ABB RobotStudio station: project_station_1_34.rspag

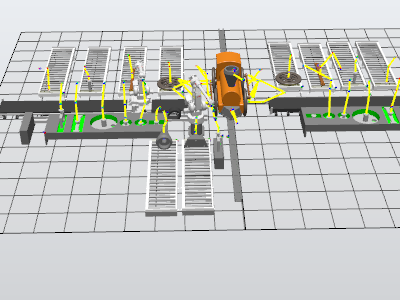
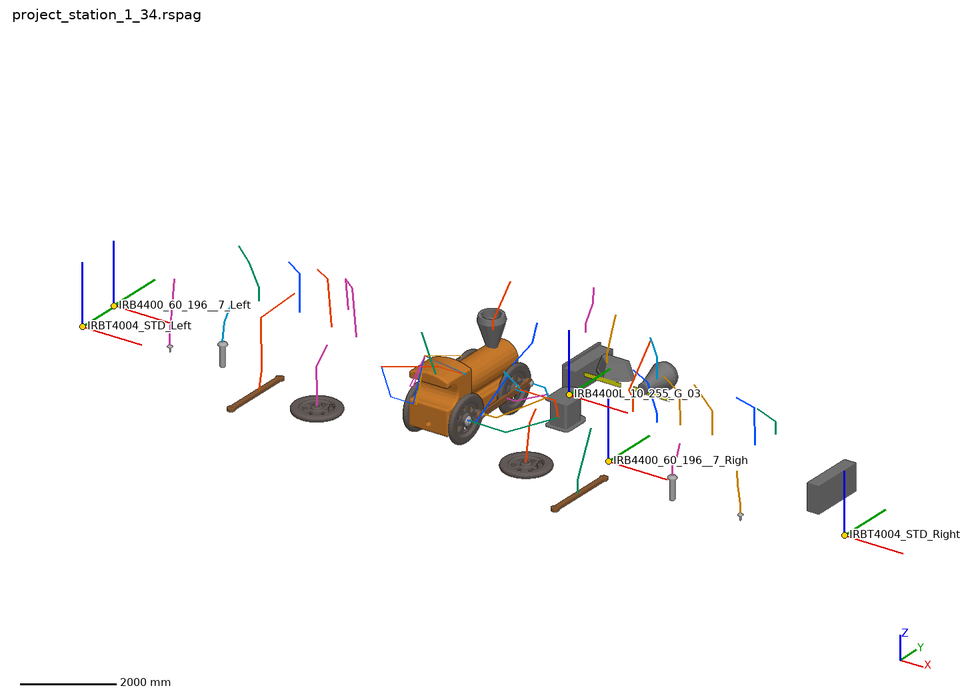
[picture v1: parts stored in the station drawn from their meshes, with robot base, taught points and paths (robot models come from the ABB library and are not in the file)]
--- station ---
Station project_station (saved by RobotStudio 24.1.10713.1)
Controller Controller2, task T_ROB1: task frame (RAPID world) sits at (1541.9, 2103.34, 619.07) mm, rotated rx 0 ry 0 rz 90 deg in the station
Controller Controller1, task T_ROB2: task frame (RAPID world) sits at (-8880.33, 560, 374.5) mm in the station
Controller Controller1, task T_ROB1: task frame (RAPID world) sits at (-8880.33, 560, 374.5) mm in the station
Controller Controller1
  mechanical unit ROB_1: IRB4400_60_196__7_Left, 6 joints, base frame (22.17, 0, 0) mm
  mechanical unit TRACK_1: IRBT4004_STD_Left, 1 joints, base frame (0, 0, 0) mm
  mechanical unit ROB_2: IRB4400_60_196__7_Right, 6 joints, base frame (17794.4, -138.17, 0) mm, rotated rx 0 ry 0 rz 180 deg
  mechanical unit TRACK_2: IRBT4004_STD_Right, 1 joints, base frame (17779.2, -146.88, 0) mm, rotated rx 0 ry 0 rz 180 deg
Controller Controller2
  mechanical unit ROB_1: IRB4400L_10_255_G_03, 6 joints, base frame (0, 0, 0) mm
Layout (positions relative to the parent item):
  - IRBT4004_STD_Right [mechanism] at (9294.37, 973.12, 0) mm, rotated rx 0 ry 0 rz 180 deg; joint values [5.175] (rad or m)
      links: Base, Link1
  - IRB4400_60_196__7_Left [mechanism, from %ABB.RobotStudio.Models.IRB4400%\IRB4400_60_196_G_03.rslib] at (-8880.33, 560, 374.5) mm; joint values [0, 0, 0, 0, 0.5236, 0] (rad or m)
  - IRB4400_60_196__7_Right [mechanism, from %ABB.RobotStudio.Models.IRB4400%\IRB4400_60_196_G_03.rslib] at (3723.87, 413.12, 374.5) mm, rotated rx 0 ry 0 rz 180 deg; joint values [-1.4312, -0.0428, -0.1313, 0, 1.1785, -0.0001] (rad or m)
  - IRBT4004_STD_Left [mechanism] at (-9275.83, 0, 0) mm; joint values [0] (rad or m)
      links: Base, Link1
  - Tool_Arm_Pin_Lift [mechanism, from Tool_geometries\my_Tool_Arm_Pin.rslib] at (-3735.45, 1947.72, 539.12) mm, rotated rx 180 ry 0 rz 180 deg
  - Tool_cow_catcher_Lift [mechanism, from Tool_geometries\my_Tool_Cow_Catcher.rslib] at (-3122.22, 1950.37, 611.02) mm, rotated rx 180 ry 0 rz 180 deg
  - Tool_Link_Right [mechanism, from Tool_geometries\my_Tool_Link.rslib] at (6128.18, 2244.28, 687.69) mm, rotated rx 180 ry -0.89 rz 180 deg
  - Tool_Stack_Right [mechanism, from Tool_geometries\my_Tool_Stack.rslib] at (733.33, 3848.22, 1135.13) mm, rotated rx 180 ry -0.01 rz -89.98 deg
  - Tool_Wheel_Right [mechanism, from Tool_geometries\my_Tool_Wheel.rslib] at (5126.19, 2141.41, 679.13) mm, rotated rx 180 ry 0 rz 180 deg
  - Tool_Axel_Pin_Lift [mechanism, from Tool_geometries\my_Too_Axel_pin.rslib] at (-4319.95, 1897.69, 635.99) mm, rotated rx 180 ry 0 rz 180 deg
  - Tool_Arm_Pin_Right [mechanism, from Tool_geometries\my_Tool_Arm_Pin.rslib] at (3680.28, 2224.13, 539.12) mm, rotated rx 180 ry 0 rz 180 deg
  - Tool_Axel_Pin_Right [mechanism, from Tool_geometries\my_Too_Axel_pin.rslib] at (4264.79, 2224.13, 633.5) mm, rotated rx 180 ry 0 rz 180 deg
  - Tool_cow_catcher_Right [mechanism, from Tool_geometries\my_Tool_Cow_Catcher.rslib] at (3068.05, 2237.38, 611.02) mm, rotated rx 180 ry 0 rz 180 deg
  - Tool_Link_Lift [mechanism, from Tool_geometries\my_Tool_Link.rslib] at (-6165.14, 1926.5, 700.28) mm, rotated rx 180 ry 0 rz 180 deg
  - Tool_Stack_Lift [mechanism, from Tool_geometries\my_Tool_Stack.rslib] at (-6789.17, 1963.76, 1135.13) mm, rotated rx 180 ry -0.01 rz 90.02 deg
  - Tool_Wheel_Lift [mechanism, from Tool_geometries\my_Tool_Wheel.rslib] at (-5181.37, 1991.55, 679.13) mm, rotated rx 180 ry 0 rz 180 deg
  - train_body [part] at (137.43, 399.25, 608.27) mm, rotated rx 0 ry 0 rz -90 deg, size 2750 x 1000 x 1362.5 mm
  - Wheel_Right_1 [part], size 1122.9 x 1119.7 x 250 mm
  - Wheel_Left_1 [part], size 1122.9 x 1119.7 x 250 mm
  - Table_tool_Right [part, from Tool_geometries\Stand_2.rslib] at (2653.05, 1565.95, 0) mm
  - Table_tool_Left [part, from Tool_geometries\Stand_2.rslib] at (-2708.23, 2555.9, 0) mm, rotated rx 0 ry 0 rz 180 deg
  - InFeeder_Right_1 [smart component, from Tool_geometries\my_InFeeder.rslib] at (2013.31, -295.59, 0) mm, rotated rx 0 ry 0 rz -90 deg
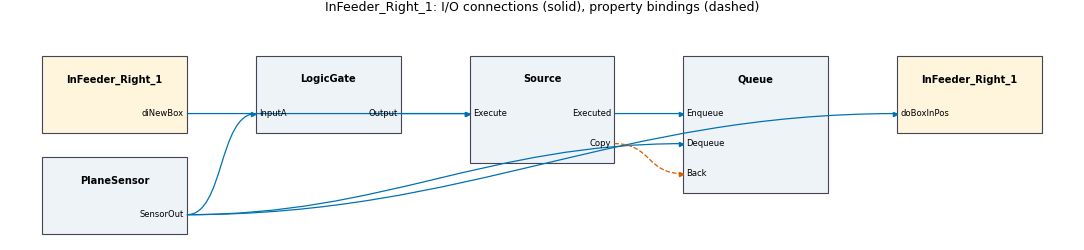
      connections:
        InFeeder_Right_1.diNewBox -> Source.Execute
        Source.Executed -> Queue.Enqueue
        PlaneSensor.SensorOut -> Queue.Dequeue
        PlaneSensor.SensorOut -> InFeeder_Right_1.doBoxInPos
        PlaneSensor.SensorOut -> LogicGate.InputA
        LogicGate.Output -> Source.Execute
        Source.Copy => Queue.Back
    - InFeeder [part, from Tool_geometries\my_InFeeder.rslib] at (-1070.62, 535.51, 0) mm
    - Source [smart component, from Components\Source.rslib] at (-1070.62, 535.51, 0) mm
        properties: Source=Wheel_Right_1; Copy=Wheel_Right_1_14; Parent=(none); Position=[0 0 0]; Orientation=[0 0 0]; Transient=false; PhysicsBehavior=-1
    - LinearMover [smart component, from Components\LinearMover.rslib] at (-1070.62, 535.51, 0) mm
        properties: Object=Queue; Direction=[0 1 0]; Speed=0.5; Reference=Global; ReferenceObject=(none)
    - Queue [smart component, from Components\Queue.rslib] at (-1070.62, 535.51, 0) mm
        properties: Back=Wheel_Right_1_14; Front=(none); Queue={1d023130-7791-4ef6-a898-f64e04810100};{8419fcdd-9884-4339-b140-c1e620e2220c};{d1e6a07f-8120-4cc8-bbc1-a0769f3691a2};{ab91239c-fc08-48bf-8341-3ec617d8a8b3}; NumberOfObjects=0
    - PlaneSensor [smart component, from Components\PlaneSensor.rslib] at (-1070.62, 535.51, 0) mm
        properties: Origin=[1.14 0.485 0.435]; Axis1=[0 0 0.1]; Axis2=[0 -0.93 0]; SensedPart=Wheel_Right_1_14; Tag=(none)
      - _sensorPart_ [part, from Tool_geometries\my_InFeeder.rslib]
    - LogicGate [smart component, from Components\LogicGate.rslib] at (-1070.62, 535.51, 0) mm
        properties: Operator=NOT; Delay=0
  - InFeeder_Right_2 [smart component, from Tool_geometries\my_InFeeder.rslib] at (3679.31, -295.59, 0) mm, rotated rx 0 ry 0 rz -90 deg
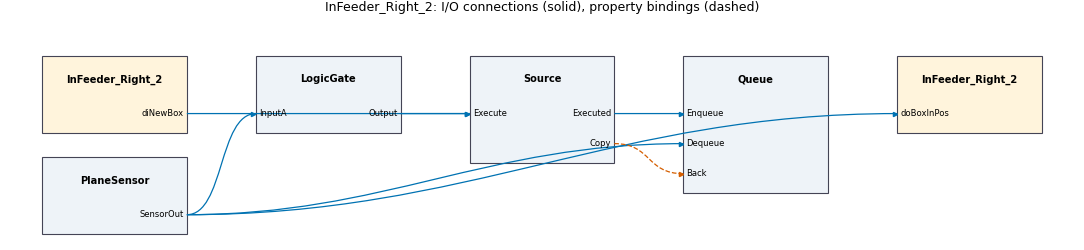
      connections:
        InFeeder_Right_2.diNewBox -> Source.Execute
        Source.Executed -> Queue.Enqueue
        PlaneSensor.SensorOut -> Queue.Dequeue
        PlaneSensor.SensorOut -> InFeeder_Right_2.doBoxInPos
        PlaneSensor.SensorOut -> LogicGate.InputA
        LogicGate.Output -> Source.Execute
        Source.Copy => Queue.Back
    - InFeeder [part, from Tool_geometries\my_InFeeder.rslib] at (-1070.62, 535.51, 0) mm
    - Source [smart component, from Components\Source.rslib] at (-1070.62, 535.51, 0) mm
        properties: Source=Link_Right_1; Copy=Link_Right_1_22; Parent=(none); Position=[0 0 0]; Orientation=[0 0 0]; Transient=false; PhysicsBehavior=-1
    - LinearMover [smart component, from Components\LinearMover.rslib] at (-1070.62, 535.51, 0) mm
        properties: Object=Queue; Direction=[0 1 0]; Speed=0.5; Reference=Global; ReferenceObject=(none)
    - Queue [smart component, from Components\Queue.rslib] at (-1070.62, 535.51, 0) mm
        properties: Back=Link_Right_1_22; Front=(none); Queue={ff46d1e0-f2c2-4271-a6c0-0c7e19cfd327};{f4dfb6bb-2350-47c6-830a-77889a19a4bb}; NumberOfObjects=0
    - PlaneSensor [smart component, from Components\PlaneSensor.rslib] at (-1070.62, 535.51, 0) mm
        properties: Origin=[1.14 0.485 0.435]; Axis1=[0 0 0.1]; Axis2=[0 -0.93 0]; SensedPart=Link_Right_1_22; Tag=(none)
      - _sensorPart_ [part, from Tool_geometries\my_InFeeder.rslib]
    - LogicGate [smart component, from Components\LogicGate.rslib] at (-1070.62, 535.51, 0) mm
        properties: Operator=NOT; Delay=0
  - InFeeder_Right_3 [smart component, from Tool_geometries\my_InFeeder.rslib] at (5345.31, -295.59, 0) mm, rotated rx 0 ry 0 rz -90 deg
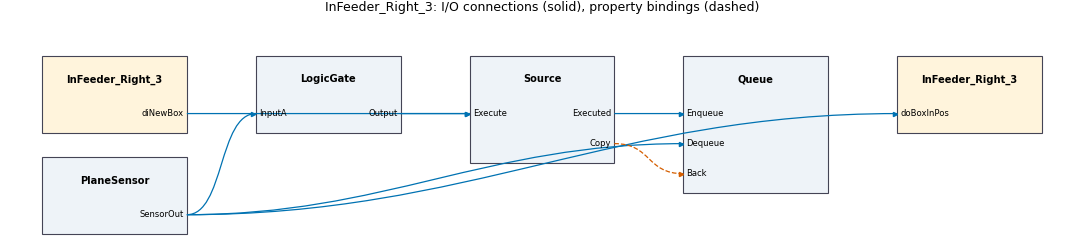
      connections:
        InFeeder_Right_3.diNewBox -> Source.Execute
        Source.Executed -> Queue.Enqueue
        PlaneSensor.SensorOut -> Queue.Dequeue
        PlaneSensor.SensorOut -> InFeeder_Right_3.doBoxInPos
        PlaneSensor.SensorOut -> LogicGate.InputA
        LogicGate.Output -> Source.Execute
        Source.Copy => Queue.Back
    - InFeeder [part, from Tool_geometries\my_InFeeder.rslib] at (-1070.62, 535.51, 0) mm
    - Source [smart component, from Components\Source.rslib] at (-1070.62, 535.51, 0) mm
        properties: Source=Axel_pin_Right_1; Copy=Axel_pin_Right_1_19; Parent=(none); Position=[0 0 0]; Orientation=[0 0 0]; Transient=false; PhysicsBehavior=-1
    - LinearMover [smart component, from Components\LinearMover.rslib] at (-1070.62, 535.51, 0) mm
        properties: Object=Queue; Direction=[0 1 0]; Speed=0.5; Reference=Global; ReferenceObject=(none)
    - Queue [smart component, from Components\Queue.rslib] at (-1070.62, 535.51, 0) mm
        properties: Back=Axel_pin_Right_1_19; Front=(none); Queue=; NumberOfObjects=0
    - PlaneSensor [smart component, from Components\PlaneSensor.rslib] at (-1070.62, 535.51, 0) mm
        properties: Origin=[1.14 0.485 0.435]; Axis1=[0 0 0.1]; Axis2=[0 -0.93 0]; SensedPart=Axel_pin_Right_1_19; Tag=(none)
      - _sensorPart_ [part, from Tool_geometries\my_InFeeder.rslib]
    - LogicGate [smart component, from Components\LogicGate.rslib] at (-1070.62, 535.51, 0) mm
        properties: Operator=NOT; Delay=0
  - InFeeder_Right_4 [smart component, from Tool_geometries\my_InFeeder.rslib] at (7011.31, -295.59, 0) mm, rotated rx 0 ry 0 rz -90 deg
      connections:
        InFeeder_Right_4.diNewBox -> Source.Execute
        Source.Executed -> Queue.Enqueue
        PlaneSensor.SensorOut -> Queue.Dequeue
        PlaneSensor.SensorOut -> InFeeder_Right_4.doBoxInPos
        PlaneSensor.SensorOut -> LogicGate.InputA
        LogicGate.Output -> Source.Execute
        Source.Copy => Queue.Back
    - InFeeder [part, from Tool_geometries\my_InFeeder.rslib] at (-1070.62, 535.51, 0) mm
    - Source [smart component, from Components\Source.rslib] at (-1070.62, 535.51, 0) mm
        properties: Source=Arm_pin_Right_1; Copy=Arm_pin_Right_1_24; Parent=(none); Position=[0 0 0]; Orientation=[0 0 0]; Transient=false; PhysicsBehavior=-1
    - LinearMover [smart component, from Components\LinearMover.rslib] at (-1070.62, 535.51, 0) mm
        properties: Object=Queue; Direction=[0 1 0]; Speed=0.5; Reference=Global; ReferenceObject=(none)
    - Queue [smart component, from Components\Queue.rslib] at (-1070.62, 535.51, 0) mm
        properties: Back=Arm_pin_Right_1_24; Front=(none); Queue=; NumberOfObjects=0
    - PlaneSensor [smart component, from Components\PlaneSensor.rslib] at (-1070.62, 535.51, 0) mm
        properties: Origin=[1.14 0.485 0.435]; Axis1=[0 0 0.1]; Axis2=[0 -0.93 0]; SensedPart=Arm_pin_Right_1_24; Tag=(none)
      - _sensorPart_ [part, from Tool_geometries\my_InFeeder.rslib]
    - LogicGate [smart component, from Components\LogicGate.rslib] at (-1070.62, 535.51, 0) mm
        properties: Operator=NOT; Delay=0
  - InFeeder_Left_1 [smart component, from Tool_geometries\my_InFeeder.rslib] at (-3038.95, -595.59, 0) mm, rotated rx 0 ry 0 rz -90 deg
      connections:
        InFeeder_Left_1.diNewBox -> Source.Execute
        Source.Executed -> Queue.Enqueue
        PlaneSensor.SensorOut -> Queue.Dequeue
        PlaneSensor.SensorOut -> InFeeder_Left_1.doBoxInPos
        PlaneSensor.SensorOut -> LogicGate.InputA
        LogicGate.Output -> Source.Execute
        Source.Copy => Queue.Back
    - InFeeder [part, from Tool_geometries\my_InFeeder.rslib] at (-1070.62, 535.51, 0) mm
    - Source [smart component, from Components\Source.rslib] at (-1070.62, 535.51, 0) mm
        properties: Source=Wheel_Left_1; Copy=Wheel_Left_1_13; Parent=(none); Position=[0 0 0]; Orientation=[0 0 0]; Transient=false; PhysicsBehavior=-1
    - LinearMover [smart component, from Components\LinearMover.rslib] at (-1070.62, 535.51, 0) mm
        properties: Object=Queue; Direction=[0 1 0]; Speed=0.5; Reference=Global; ReferenceObject=(none)
    - Queue [smart component, from Components\Queue.rslib] at (-1070.62, 535.51, 0) mm
        properties: Back=Wheel_Left_1_13; Front=(none); Queue=; NumberOfObjects=0
    - PlaneSensor [smart component, from Components\PlaneSensor.rslib] at (-1070.62, 535.51, 0) mm
        properties: Origin=[1.14 0.485 0.435]; Axis1=[0 0 0.1]; Axis2=[0 -0.93 0]; SensedPart=Wheel_Left_1_13; Tag=(none)
      - _sensorPart_ [part, from Tool_geometries\my_InFeeder.rslib]
    - LogicGate [smart component, from Components\LogicGate.rslib] at (-1070.62, 535.51, 0) mm
        properties: Operator=NOT; Delay=0
  - InFeeder_Left_2 [smart component, from Tool_geometries\my_InFeeder.rslib] at (-4426.95, -445.59, 0) mm, rotated rx 0 ry 0 rz -90 deg
      connections:
        InFeeder_Left_2.diNewBox -> Source.Execute
        Source.Executed -> Queue.Enqueue
        PlaneSensor.SensorOut -> Queue.Dequeue
        PlaneSensor.SensorOut -> InFeeder_Left_2.doBoxInPos
        PlaneSensor.SensorOut -> LogicGate.InputA
        LogicGate.Output -> Source.Execute
        Source.Copy => Queue.Back
    - InFeeder [part, from Tool_geometries\my_InFeeder.rslib] at (-1070.62, 535.51, 0) mm
    - Source [smart component, from Components\Source.rslib] at (-1070.62, 535.51, 0) mm
        properties: Source=Link_Left_1; Copy=Link_Left_1_18; Parent=(none); Position=[0 0 0]; Orientation=[0 0 0]; Transient=false; PhysicsBehavior=-1
    - LinearMover [smart component, from Components\LinearMover.rslib] at (-1070.62, 535.51, 0) mm
        properties: Object=Queue; Direction=[0 1 0]; Speed=0.5; Reference=Global; ReferenceObject=(none)
    - Queue [smart component, from Components\Queue.rslib] at (-1070.62, 535.51, 0) mm
        properties: Back=Link_Left_1_18; Front=(none); Queue={1ff3d472-21b5-4bb2-8564-f6cc722a728c}; NumberOfObjects=0
    - PlaneSensor [smart component, from Components\PlaneSensor.rslib] at (-1070.62, 535.51, 0) mm
        properties: Origin=[1.14 0.485 0.435]; Axis1=[0 0 0.1]; Axis2=[0 -0.93 0]; SensedPart=Link_Left_1_18; Tag=(none)
      - _sensorPart_ [part, from Tool_geometries\my_InFeeder.rslib]
    - LogicGate [smart component, from Components\LogicGate.rslib] at (-1070.62, 535.51, 0) mm
        properties: Operator=NOT; Delay=0
  - InFeeder_Left_3 [smart component, from Tool_geometries\my_InFeeder.rslib] at (-5792.95, -595.59, 0) mm, rotated rx 0 ry 0 rz -90 deg
      connections:
        InFeeder_Left_3.diNewBox -> Source.Execute
        Source.Executed -> Queue.Enqueue
        PlaneSensor.SensorOut -> Queue.Dequeue
        PlaneSensor.SensorOut -> InFeeder_Left_3.doBoxInPos
        PlaneSensor.SensorOut -> LogicGate.InputA
        LogicGate.Output -> Source.Execute
        Source.Copy => Queue.Back
    - InFeeder [part, from Tool_geometries\my_InFeeder.rslib] at (-1070.62, 535.51, 0) mm
    - Source [smart component, from Components\Source.rslib] at (-1070.62, 535.51, 0) mm
        properties: Source=Axel_pin_Left_1; Copy=Axel_pin_Left_1_16; Parent=(none); Position=[0 0 0]; Orientation=[0 0 0]; Transient=false; PhysicsBehavior=-1
    - LinearMover [smart component, from Components\LinearMover.rslib] at (-1070.62, 535.51, 0) mm
        properties: Object=Queue; Direction=[0 1 0]; Speed=0.5; Reference=Global; ReferenceObject=(none)
    - Queue [smart component, from Components\Queue.rslib] at (-1070.62, 535.51, 0) mm
        properties: Back=Axel_pin_Left_1_16; Front=(none); Queue={9023f18c-56cf-4535-be10-c416e51bdbb7};{c60a748b-6081-462f-837c-dfeccbfd19db};{920b546f-ac67-4257-bb71-08cb4a795493}; NumberOfObjects=0
    - PlaneSensor [smart component, from Components\PlaneSensor.rslib] at (-1070.62, 535.51, 0) mm
        properties: Origin=[1.14 0.485 0.435]; Axis1=[0 0 0.1]; Axis2=[0 -0.93 0]; SensedPart=Axel_pin_Left_1_16; Tag=(none)
      - _sensorPart_ [part, from Tool_geometries\my_InFeeder.rslib]
    - LogicGate [smart component, from Components\LogicGate.rslib] at (-1070.62, 535.51, 0) mm
        properties: Operator=NOT; Delay=0
  - InFeeder_Left_4 [smart component, from Tool_geometries\my_InFeeder.rslib] at (-7158.95, -595.59, 0) mm, rotated rx 0 ry 0 rz -90 deg
      connections:
        InFeeder_Left_4.diNewBox -> Source.Execute
        Source.Executed -> Queue.Enqueue
        PlaneSensor.SensorOut -> Queue.Dequeue
        PlaneSensor.SensorOut -> InFeeder_Left_4.doBoxInPos
        PlaneSensor.SensorOut -> LogicGate.InputA
        LogicGate.Output -> Source.Execute
        Source.Copy => Queue.Back
    - InFeeder [part, from Tool_geometries\my_InFeeder.rslib] at (-1070.62, 535.51, 0) mm
    - Source [smart component, from Components\Source.rslib] at (-1070.62, 535.51, 0) mm
        properties: Source=Arm_pin_Left_1; Copy=Arm_pin_Left_1_21; Parent=(none); Position=[0 0 0]; Orientation=[0 0 0]; Transient=false; PhysicsBehavior=-1
    - LinearMover [smart component, from Components\LinearMover.rslib] at (-1070.62, 535.51, 0) mm
        properties: Object=Queue; Direction=[0 1 0]; Speed=0.5; Reference=Global; ReferenceObject=(none)
    - Queue [smart component, from Components\Queue.rslib] at (-1070.62, 535.51, 0) mm
        properties: Back=Arm_pin_Left_1_21; Front=(none); Queue=; NumberOfObjects=0
    - PlaneSensor [smart component, from Components\PlaneSensor.rslib] at (-1070.62, 535.51, 0) mm
        properties: Origin=[1.14 0.485 0.435]; Axis1=[0 0 0.1]; Axis2=[0 -0.93 0]; SensedPart=Arm_pin_Left_1_21; Tag=(none)
      - _sensorPart_ [part, from Tool_geometries\my_InFeeder.rslib]
    - LogicGate [smart component, from Components\LogicGate.rslib] at (-1070.62, 535.51, 0) mm
        properties: Operator=NOT; Delay=0
  - Link_Right_1 [part] at (0, 300, 0) mm, size 186.8 x 1937.5 x 62.5 mm
  - train_tool_test [mechanism, from Tool_geometries\Train_Tool.rslib] at (0, 6532.17, 0) mm, rotated rx 0 ry 0 rz -90 deg; joint values [-0.5587, 0] (rad or m)
  - SC_AttachTool_Right [smart component] at (7697.63, 413.12, 2024.5) mm, rotated rx 180 ry 60 rz 0 deg
      signals: DI diAttachTool
      connections:
        SC_AttachTool_Right.diAttachTool -> ClosestObject.Execute
        ClosestObject.Executed -> Attacher.Execute
        SC_AttachTool_Right.diAttachTool -> LogicGate.InputA
        LogicGate.Output -> Detacher.Execute
        ClosestObject.ClosestObject => Attacher.Child
        Attacher.Child => Detacher.Child
    - Attacher [smart component, from Components\Attacher.rslib]
        properties: Parent=IRB4400_60_196__7_Right; Flange=0; Child=Tool_Arm_Pin_Right; Mount=false; Offset=[0 0 0]; Orientation=[0 0 0]
    - Detacher [smart component, from Components\Detacher.rslib]
        properties: Child=Tool_Arm_Pin_Right; KeepPosition=true
    - ClosestObject [smart component, from Components\ClosestObject.rslib]
        properties: ReferenceObject=IRB4400_60_196__7_Right; ReferencePoint=[7.697628 0.41312 2.0245]; RootObject=(none); ClosestObject=Tool_Arm_Pin_Right; ClosestPart=Tool_Arm_pin; Distance=0
    - LogicGate [smart component, from Components\LogicGate.rslib]
        properties: Operator=NOT; Delay=0
  - Axel_pin_Left_1 [part] at (1364.35, 150, 0) mm, size 211 x 211 x 562.7 mm
  - Arm_pin_Left_1 [part], size 126 x 125.8 x 162.5 mm
  - Link_Left_1 [part], size 186.8 x 1937.5 x 62.5 mm
  - SC_AttachTool_left [smart component] at (-8447.37, 1113.95, 2155.74) mm, rotated rx 180 ry 60 rz -130.35 deg
      signals: DI diAT_Left
      connections:
        SC_AttachTool_left.diAT_Left -> ClosestObject.Execute
        ClosestObject.Executed -> Attacher.Execute
        SC_AttachTool_left.diAT_Left -> LogicGate.InputA
        LogicGate.Output -> Detacher.Execute
        ClosestObject.ClosestObject => Attacher.Child
        Attacher.Child => Detacher.Child
    - Attacher [smart component, from Components\Attacher.rslib]
        properties: Parent=IRB4400_60_196__7_Left; Flange=0; Child=Tool_Arm_Pin_Lift; Mount=false; Offset=[0 0 0]; Orientation=[0 0 0]
    - Detacher [smart component, from Components\Detacher.rslib]
        properties: Child=Tool_Arm_Pin_Lift; KeepPosition=true
    - ClosestObject [smart component, from Components\ClosestObject.rslib]
        properties: ReferenceObject=IRB4400_60_196__7_Left; ReferencePoint=[-7.679085 0.56 2.0245]; RootObject=(none); ClosestObject=Tool_Arm_Pin_Lift; ClosestPart=Tool_Arm_pin; Distance=0
    - LogicGate [smart component, from Components\LogicGate.rslib]
        properties: Operator=NOT; Delay=0
  - Axel_pin_Right_1 [part], size 211 x 211 x 562.7 mm
  - Arm_pin_Right_1 [part], size 126 x 125.8 x 162.5 mm
  - RobotStand2400H620 [part] at (1512.32, 2162.24, 0) mm, size 600 x 830 x 620 mm
  - IRB4400L_10_255_G_03 [mechanism, from %ABB.RobotStudio.Models.IRB4400%\IRB4400L_10_255_G_03.rslib] at (1541.9, 2103.34, 619.07) mm, rotated rx 0 ry 0 rz 90 deg; joint values [0.3142, 0, 0, 0, 0.9774, 0] (rad or m)
  - SC_InFeeder [smart component, from Solutions\SC_InFeeder.rslib] at (2782.92, 2208.74, 0) mm, rotated rx 0 ry 0 rz 90 deg
      connections:
        SC_InFeeder.diNewBox -> Source.Execute
        Source.Executed -> Queue.Enqueue
        PlaneSensor.SensorOut -> Queue.Dequeue
        PlaneSensor.SensorOut -> SC_InFeeder.doBoxInPos
        PlaneSensor.SensorOut -> LogicGate.InputA
        LogicGate.Output -> Source.Execute
        Source.Copy => Queue.Back
    - InFeeder [part, from Solutions\SC_InFeeder.rslib]
    - Source [smart component, from Components\Source.rslib]
        properties: Source=Stack_tutorial; Copy=Stack_tutorial_26; Parent=(none); Position=[0 0 0]; Orientation=[0 0 0]; Transient=false; PhysicsBehavior=-1
    - LinearMover [smart component, from Components\LinearMover.rslib]
        properties: Object=Queue; Direction=[0 -1 0]; Speed=0.5; Reference=Global; ReferenceObject=(none)
    - Queue [smart component, from Components\Queue.rslib]
        properties: Back=Stack_tutorial_26; Front=(none); Queue=; NumberOfObjects=0
    - PlaneSensor [smart component, from Components\PlaneSensor.rslib]
        properties: Origin=[1.14 0.485 0.435]; Axis1=[0 0 0.1]; Axis2=[0 -0.93 0]; SensedPart=Stack_tutorial_26; Tag=(none)
      - _sensorPart_ [part], size 0 x 930 x 100 mm
    - LogicGate [smart component, from Components\LogicGate.rslib]
        properties: Operator=NOT; Delay=0
  - SC_InFeeder_1 [smart component, from Solutions\SC_InFeeder.rslib] at (1551.58, 2174.69, 0) mm, rotated rx 0 ry 0 rz 90 deg
      connections:
        SC_InFeeder_1.diNewBox -> Source.Execute
        Source.Executed -> Queue.Enqueue
        PlaneSensor.SensorOut -> Queue.Dequeue
        PlaneSensor.SensorOut -> SC_InFeeder_1.doBoxInPos
        PlaneSensor.SensorOut -> LogicGate.InputA
        LogicGate.Output -> Source.Execute
        Source.Copy => Queue.Back
    - InFeeder [part, from Solutions\SC_InFeeder.rslib]
    - Source [smart component, from Components\Source.rslib]
        properties: Source=Cow_Catcher; Copy=Cow_Catcher_25; Parent=(none); Position=[0 0 0]; Orientation=[0 0 0]; Transient=false; PhysicsBehavior=-1
    - LinearMover [smart component, from Components\LinearMover.rslib]
        properties: Object=Queue; Direction=[0 -1 0]; Speed=0.5; Reference=Global; ReferenceObject=(none)
    - Queue [smart component, from Components\Queue.rslib]
        properties: Back=Cow_Catcher_25; Front=(none); Queue=; NumberOfObjects=0
    - PlaneSensor [smart component, from Components\PlaneSensor.rslib]
        properties: Origin=[1.14 0.485 0.435]; Axis1=[0 0 0.1]; Axis2=[0 -0.93 0]; SensedPart=Cow_Catcher_25; Tag=(none)
      - _sensorPart_ [part], size 0 x 930 x 100 mm
    - LogicGate [smart component, from Components\LogicGate.rslib]
        properties: Operator=NOT; Delay=0
  - Cow_Catcher [part], size 900 x 562.5 x 375 mm
  - Stack_tutorial [part], size 625 x 875 x 623.8 mm
  - SmartComponent_1 [smart component] at (1001.89, 3765.34, 2268.6) mm, rotated rx -180 ry 34 rz -72 deg
      signals: DI di_Rob3_at_tool
      connections:
        SmartComponent_1.di_Rob3_at_tool -> ClosestObject.Execute
        ClosestObject.Executed -> Attacher.Execute
        SmartComponent_1.di_Rob3_at_tool -> LogicGate.InputA
        LogicGate.Output -> Detacher.Execute
        ClosestObject.ClosestObject => Attacher.Child
        Attacher.Child => Detacher.Child
    - Attacher [smart component, from Components\Attacher.rslib]
        properties: Parent=IRB4400L_10_255_G_03; Flange=0; Child=Tool_Stack_Right; Mount=false; Offset=[0 0 0]; Orientation=[0 0 0]
    - Detacher [smart component, from Components\Detacher.rslib]
        properties: Child=Tool_Stack_Right; KeepPosition=true
    - ClosestObject [smart component, from Components\ClosestObject.rslib] at (0, 0.07, 0.19) mm, rotated rx 0 ry 0 rz 0.01 deg
        properties: ReferenceObject=IRB4400L_10_255_G_03; ReferencePoint=[1.623149 3.935855 2.269225]; RootObject=(none); ClosestObject=Tool_Stack_Right; ClosestPart=Tool_Stack_tutorial; Distance=0
    - LogicGate [smart component, from Components\LogicGate.rslib]
        properties: Operator=NOT; Delay=0
  - Tool_Stack [mechanism, from Tool_geometries\my_Tool_Stack.rslib] at (6727.73, 2146.19, 1135.13) mm, rotated rx 180 ry -0.01 rz -89.98 deg
  - Part_1 [part] at (7983.1, 1490.43, 0) mm, size 300 x 1350 x 650 mm
  - Part_10 [part] at (543.39, 3269.91, 0) mm, size 348.3 x 1331.4 x 570 mm
  - Axel_pin_Left_1_1 [part] at (501.33, -5711.63, 5481.38) mm, rotated rx 90 ry 0 rz -90 deg, size 211 x 211 x 562.7 mm
  - Arm_pin_Left_1_2 [part] at (-187.19, 6322.39, -3373.2) mm, rotated rx -88 ry -0.94 rz 89.66 deg, size 126 x 125.8 x 162.5 mm
  - Stack_tutorial_3 [part] at (191.58, -1196.82, -5198.95) mm, rotated rx 89.7 ry -2.42 rz 106.93 deg, size 625 x 875 x 623.8 mm
  - Cow_Catcher_4 [part] at (2358.03, 9034.46, -915.07) mm, rotated rx 8.93 ry 3.16 rz 175.56 deg, size 900 x 562.5 x 375 mm
  - Link_Left_1_5 [part] at (-36.44, -4252.23, -2713.27) mm, rotated rx 99.73 ry 90 rz -80.27 deg, size 186.8 x 1937.5 x 62.5 mm
  - Wheel_Right_1_6 [part] at (297.93, -1737.55, 5267.12) mm, rotated rx 91.04 ry -5.67 rz 89.75 deg, size 1122.9 x 1119.7 x 250 mm
  - Link_Right_1_7 [part] at (436, -3607.65, -3457.42) mm, rotated rx -88.02 ry -88 rz -91.77 deg, size 186.8 x 1937.5 x 62.5 mm
  - Axel_pin_Right_1_8 [part] at (-147.05, -5745.67, 2902.14) mm, rotated rx 90 ry -20 rz 90 deg, size 211 x 211 x 562.7 mm
  - Arm_pin_Right_1_9 [part] at (1185.67, -6952.34, -808.64) mm, rotated rx 88.67 ry -40.63 rz 96.05 deg, size 126 x 125.8 x 162.5 mm
  - Wheel_Left_1_10 [part] at (65.04, 4540.99, 1028.75) mm, rotated rx -90 ry -62 rz 90 deg, size 1122.9 x 1119.7 x 250 mm
  - Wheel_Left_1_11 [part] at (65.04, 6286.67, 1028.75) mm, rotated rx -90 ry -62 rz 90 deg, size 1122.9 x 1119.7 x 250 mm
  - Wheel_Right_1_12 [part] at (374.22, -3437.13, 5308.69) mm, rotated rx 93.56 ry -5.2 rz 87.1 deg, size 1122.9 x 1119.7 x 250 mm
  - Wheel_Left_1_13 [part] at (0, 3132, 0) mm, size 1122.9 x 1119.7 x 250 mm
  - Wheel_Right_1_14 [part] at (0, 3756, 0) mm, size 1122.9 x 1119.7 x 250 mm
  - Axel_pin_Left_1_15 [part] at (501.09, -3965.51, 5481.38) mm, rotated rx 90 ry 0 rz -90 deg, size 211 x 211 x 562.7 mm
  - Axel_pin_Left_1_16 [part] at (0, 3900, 0) mm, size 211 x 211 x 562.7 mm
  - Axel_pin_Right_1_17 [part] at (-152.97, -7511.91, 2881.93) mm, rotated rx 90 ry -20 rz 90 deg, size 211 x 211 x 562.7 mm
  - Link_Left_1_18 [part] at (0, 3312, 0) mm, size 186.8 x 1937.5 x 62.5 mm
  - Axel_pin_Right_1_19 [part] at (0, 3900, 0) mm, size 211 x 211 x 562.7 mm
  - Arm_pin_Left_1_20 [part] at (-187.19, 8072.39, -3373.2) mm, rotated rx -88 ry -0.94 rz 89.66 deg, size 126 x 125.8 x 162.5 mm
  - Arm_pin_Left_1_21 [part] at (0, 3960, 0) mm, size 126 x 125.8 x 162.5 mm
  - Link_Right_1_22 [part] at (0, 3132, 0) mm, size 186.8 x 1937.5 x 62.5 mm
  - Arm_pin_Right_1_23 [part] at (1192.07, -8711.93, -803.85) mm, rotated rx 88.67 ry -40.63 rz 96.05 deg, size 126 x 125.8 x 162.5 mm
  - Arm_pin_Right_1_24 [part] at (0, 3912, 0) mm, size 126 x 125.8 x 162.5 mm
  - Cow_Catcher_25 [part] at (0, -3876, 0) mm, size 900 x 562.5 x 375 mm
  - Stack_tutorial_26 [part] at (0, -3564, 0) mm, size 625 x 875 x 623.8 mm
Attachment: IRB4400_60_196__7_Left is attached to IRBT4004_STD_Left / Link1
Attachment: stand_tool_Right is attached to Table_tool_Right
Attachment: stand_tool_Left is attached to Table_tool_Left
Attachment: Tool_cow_catcher_Lift is attached to Table_tool_Left
Attachment: InFeWOb_Right_1 is attached to InFeeder
Attachment: InFeWOb_Right_2 is attached to InFeeder
Attachment: InFeWOb_Right_3 is attached to InFeeder
Attachment: InFeWOb_Right_4 is attached to InFeeder
Attachment: Link_Right_1 is attached to InFeeder_Right_2
Attachment: InFeWOb_Lift_1 is attached to InFeeder
Attachment: InFeWOb_Lift_3 is attached to InFeeder
Attachment: InFeWOb_Lift_2 is attached to InFeeder
Attachment: InFeWOb_Lift_4 is attached to InFeeder
Attachment: TrRiFcWOb is attached to train_body
Attachment: TrLeFcWob is attached to train_body
Attachment: Arm_pin_Left_1 is attached to InFeeder_Left_3
Attachment: Axel_pin_Left_1 is attached to InFeeder_Left_2
Attachment: Link_Left_1 is attached to InFeeder_Left_4
Attachment: Wheel_Left_1 is attached to InFeeder_Left_1
Attachment: Axel_pin_Right_1 is attached to InFeeder_Right_3
Attachment: Arm_pin_Right_1 is attached to InFeeder_Right_4
Attachment: IRB4400_60_196__7_Right is attached to IRBT4004_STD_Right / Link1
Attachment: WokOb_feed_1_Caw is attached to InFeeder
Attachment: WokOb_feed is attached to InFeeder
Attachment: WokOb_tarin_Front is attached to train_body
Attachment: WokOb_Train_Top is attached to train_body
Attachment: SmartComponent_1 is attached to IRB4400L_10_255_G_03 / Link6
Attachment: Cow_Catcher is attached to SC_InFeeder_1
Attachment: IRB4400L_10_255_G_03 is attached to RobotStand2400H620
Attachment: WorOb_Stacl_Rb3 is attached to Part_10
EventTableEntry 6118: Group=, Trigger=diAttachTool 6119, Actions=[EventTableActionAttach 6120], Comment=, ActivationMode=2, Cyclic=false
EventTableTriggerIO 6119: IOValue=[1], IRC5Controller=? -1, Operator=0, SignalSource=Controller1 3715
EventTableActionAttach 6120: AttachmentParent=IRB4400_60_196__7_Right 3583, AttachmentChild=? -1, MountObject=false, Offset=[X=1, Y=0, Z=0, W=0, X=0, Y=1, Z=0, W=0, X=0, Y=0, Z=1, W=0, X=0, Y=0, Z=0, W=1], FlangeIndext=0, FindNearest=true
EventTableEntry 6121: Group=, Trigger=diAttachTool 6122, Actions=[EventTableActionDetach 6123], Comment=, ActivationMode=2, Cyclic=false
EventTableTriggerIO 6122: IOValue=[0], IRC5Controller=? -1, Operator=0, SignalSource=Controller1 3715
EventTableActionDetach 6123: AttachmentParent=IRB4400_60_196__7_Right 3583, AttachmentChild=? -1
EventTableEntry 8584: Group=, Trigger=doAttachTool 8585, Actions=[EventTableActionAttach 8586], Comment=, ActivationMode=2, Cyclic=false
EventTableTriggerIO 8585: IOValue=[1], IRC5Controller=? -1, Operator=0, SignalSource=Controller1 3715
EventTableActionAttach 8586: AttachmentParent=IRB4400_60_196__7_Left 2378, AttachmentChild=? -1, MountObject=false, Offset=[X=1, Y=0, Z=0, W=0, X=0, Y=1, Z=0, W=0, X=0, Y=0, Z=1, W=0, X=0, Y=0, Z=0, W=1], FlangeIndext=0, FindNearest=true
EventTableEntry 8587: Group=, Trigger=doAttachTool 8588, Actions=[EventTableActionDetach 8589], Comment=, ActivationMode=2, Cyclic=false
EventTableTriggerIO 8588: IOValue=[0], IRC5Controller=? -1, Operator=0, SignalSource=Controller1 3715
EventTableActionDetach 8589: AttachmentParent=IRB4400_60_196__7_Left 2378, AttachmentChild=? -1
EventTableEntry 10457: Group=, Trigger=doAtWhRi 10458, Actions=[EventTableActionAttach 10459], Comment=, ActivationMode=2, Cyclic=false
EventTableTriggerIO 10458: IOValue=[1], IRC5Controller=? -1, Operator=0, SignalSource=Controller1 3715
EventTableActionAttach 10459: AttachmentParent=Tool_Wheel_Right 3673, AttachmentChild=? -1, MountObject=false, Offset=[X=1, Y=0, Z=0, W=0, X=0, Y=1, Z=0, W=0, X=0, Y=0, Z=1, W=0, X=0, Y=0, Z=0, W=1], FlangeIndext=0, FindNearest=true
EventTableEntry 10462: Group=, Trigger=doAtWhRi 10463, Actions=[EventTableActionDetach 10464], Comment=, ActivationMode=2, Cyclic=false
EventTableTriggerIO 10463: IOValue=[0], IRC5Controller=? -1, Operator=0, SignalSource=Controller1 3715
EventTableActionDetach 10464: AttachmentParent=Tool_Wheel_Right 3673, AttachmentChild=? -1
EventTableEntry 10559: Group=, Trigger=Att_link 10560, Actions=[EventTableActionAttach 10561], Comment=, ActivationMode=2, Cyclic=false
EventTableTriggerIO 10560: IOValue=[1], IRC5Controller=? -1, Operator=0, SignalSource=Controller1 3715
EventTableActionAttach 10561: AttachmentParent=Tool_Link_Right 3667, AttachmentChild=? -1, MountObject=false, Offset=[X=1, Y=0, Z=0, W=0, X=0, Y=1, Z=0, W=0, X=0, Y=0, Z=1, W=0, X=0, Y=0, Z=0, W=1], FlangeIndext=0, FindNearest=true
EventTableEntry 10562: Group=, Trigger=Att_link 10563, Actions=[EventTableActionDetach 10564], Comment=, ActivationMode=2, Cyclic=false
EventTableTriggerIO 10563: IOValue=[0], IRC5Controller=? -1, Operator=0, SignalSource=Controller1 3715
EventTableActionDetach 10564: AttachmentParent=Tool_Link_Right 3667, AttachmentChild=? -1
EventTableEntry 13658: Group=, Trigger=doAt_Wh_Left 13659, Actions=[EventTableActionAttach 13660], Comment=, ActivationMode=2, Cyclic=false
EventTableTriggerIO 13659: IOValue=[1], IRC5Controller=? -1, Operator=0, SignalSource=Controller1 3715
EventTableActionAttach 13660: AttachmentParent=Tool_Wheel_Lift 3694, AttachmentChild=? -1, MountObject=false, Offset=[X=1, Y=0, Z=0, W=0, X=0, Y=1, Z=0, W=0, X=0, Y=0, Z=1, W=0, X=0, Y=0, Z=0, W=1], FlangeIndext=0, FindNearest=true
EventTableEntry 13661: Group=, Trigger=doAt_Wh_Left 13662, Actions=[EventTableActionDetach 13663], Comment=, ActivationMode=2, Cyclic=false
EventTableTriggerIO 13662: IOValue=[0], IRC5Controller=? -1, Operator=0, SignalSource=Controller1 3715
EventTableActionDetach 13663: AttachmentParent=Tool_Wheel_Lift 3694, AttachmentChild=? -1
EventTableEntry 13664: Group=, Trigger=doAt_Link_Left 13665, Actions=[EventTableActionAttach 13666], Comment=, ActivationMode=2, Cyclic=false
EventTableTriggerIO 13665: IOValue=[1], IRC5Controller=? -1, Operator=0, SignalSource=Controller1 3715
EventTableActionAttach 13666: AttachmentParent=Tool_Link_Lift 3688, AttachmentChild=? -1, MountObject=false, Offset=[X=1, Y=0, Z=0, W=0, X=0, Y=1, Z=0, W=0, X=0, Y=0, Z=1, W=0, X=0, Y=0, Z=0, W=1], FlangeIndext=0, FindNearest=true
EventTableEntry 13667: Group=, Trigger=doAt_Link_Left 13668, Actions=[EventTableActionDetach 13669], Comment=, ActivationMode=2, Cyclic=false
EventTableTriggerIO 13668: IOValue=[0], IRC5Controller=? -1, Operator=0, SignalSource=Controller1 3715
EventTableActionDetach 13669: AttachmentParent=Tool_Link_Lift 3688, AttachmentChild=? -1
EventTableEntry 13670: Group=, Trigger=doAt_AxelP_Left 13671, Actions=[EventTableActionAttach 13672], Comment=, ActivationMode=2, Cyclic=false
EventTableTriggerIO 13671: IOValue=[1], IRC5Controller=? -1, Operator=0, SignalSource=Controller1 3715
EventTableActionAttach 13672: AttachmentParent=Tool_Axel_Pin_Lift 3676, AttachmentChild=? -1, MountObject=false, Offset=[X=1, Y=0, Z=0, W=0, X=0, Y=1, Z=0, W=0, X=0, Y=0, Z=1, W=0, X=0, Y=0, Z=0, W=1], FlangeIndext=0, FindNearest=true
EventTableEntry 13673: Group=, Trigger=doAt_AxelP_Left 13674, Actions=[EventTableActionDetach 13675], Comment=, ActivationMode=2, Cyclic=false
EventTableTriggerIO 13674: IOValue=[0], IRC5Controller=? -1, Operator=0, SignalSource=Controller1 3715
EventTableActionDetach 13675: AttachmentParent=Tool_Axel_Pin_Lift 3676, AttachmentChild=? -1
EventTableEntry 13676: Group=, Trigger=doAt_Arm_Left 13677, Actions=[EventTableActionAttach 13678], Comment=, ActivationMode=2, Cyclic=false
EventTableTriggerIO 13677: IOValue=[1], IRC5Controller=? -1, Operator=0, SignalSource=Controller1 3715
EventTableActionAttach 13678: AttachmentParent=Tool_Arm_Pin_Lift 3661, AttachmentChild=? -1, MountObject=false, Offset=[X=1, Y=0, Z=0, W=0, X=0, Y=1, Z=0, W=0, X=0, Y=0, Z=1, W=0, X=0, Y=0, Z=0, W=1], FlangeIndext=0, FindNearest=true
EventTableEntry 13679: Group=, Trigger=doAt_Arm_Left 13680, Actions=[EventTableActionDetach 13681], Comment=, ActivationMode=2, Cyclic=false
EventTableTriggerIO 13680: IOValue=[0], IRC5Controller=? -1, Operator=0, SignalSource=Controller1 3715
EventTableActionDetach 13681: AttachmentParent=Tool_Arm_Pin_Lift 3661, AttachmentChild=? -1
EventTableTriggerIO 14352: IOValue=[1], IRC5Controller=? -1, Operator=0, SignalSource=Controller1 3715
EventTableTriggerIO 14353: IOValue=[0], IRC5Controller=? -1, Operator=0, SignalSource=Controller1 3715
EventTableTriggerIO 14354: IOValue=[1], IRC5Controller=? -1, Operator=0, SignalSource=Controller1 3715
EventTableTriggerIO 14355: IOValue=[0], IRC5Controller=? -1, Operator=0, SignalSource=Controller1 3715
EventTableTriggerIO 14356: IOValue=[1], IRC5Controller=? -1, Operator=0, SignalSource=Controller1 3715
EventTableTriggerIO 14357: IOValue=[0], IRC5Controller=? -1, Operator=0, SignalSource=Controller1 3715
EventTableTriggerIO 14358: IOValue=[1], IRC5Controller=? -1, Operator=0, SignalSource=Controller1 3715
EventTableTriggerIO 14359: IOValue=[0], IRC5Controller=? -1, Operator=0, SignalSource=Controller1 3715
EventTableTriggerIO 14360: IOValue=[1], IRC5Controller=? -1, Operator=0, SignalSource=Controller1 3715
EventTableTriggerIO 14361: IOValue=[0], IRC5Controller=? -1, Operator=0, SignalSource=Controller1 3715
EventTableTriggerIO 14362: IOValue=[1], IRC5Controller=? -1, Operator=0, SignalSource=Controller1 3715
EventTableTriggerIO 14363: IOValue=[0], IRC5Controller=? -1, Operator=0, SignalSource=Controller1 3715
EventTableTriggerIO 14364: IOValue=[1], IRC5Controller=? -1, Operator=0, SignalSource=Controller1 3715
EventTableTriggerIO 14365: IOValue=[0], IRC5Controller=? -1, Operator=0, SignalSource=Controller1 3715
EventTableTriggerIO 14366: IOValue=[1], IRC5Controller=? -1, Operator=0, SignalSource=Controller1 3715
EventTableTriggerIO 14367: IOValue=[0], IRC5Controller=? -1, Operator=0, SignalSource=Controller1 3715
EventTableEntry 16109: Group=, Trigger=doAt_AxelP_Right 16110, Actions=[EventTableActionAttach 16111], Comment=, ActivationMode=2, Cyclic=false
EventTableTriggerIO 16110: IOValue=[1], IRC5Controller=? -1, Operator=0, SignalSource=Controller1 3715
EventTableActionAttach 16111: AttachmentParent=Tool_Axel_Pin_Right 3682, AttachmentChild=? -1, MountObject=false, Offset=[X=1, Y=0, Z=0, W=0, X=0, Y=1, Z=0, W=0, X=0, Y=0, Z=1, W=0, X=0, Y=0, Z=0, W=1], FlangeIndext=0, FindNearest=true
EventTableEntry 16112: Group=, Trigger=doAt_AxelP_Right 16113, Actions=[EventTableActionDetach 16114], Comment=, ActivationMode=2, Cyclic=false
EventTableTriggerIO 16113: IOValue=[0], IRC5Controller=? -1, Operator=0, SignalSource=Controller1 3715
EventTableActionDetach 16114: AttachmentParent=Tool_Axel_Pin_Right 3682, AttachmentChild=? -1
EventTableEntry 16115: Group=, Trigger=doAt_ArmP_Right 16116, Actions=[EventTableActionAttach 16117], Comment=, ActivationMode=2, Cyclic=false
EventTableTriggerIO 16116: IOValue=[1], IRC5Controller=? -1, Operator=0, SignalSource=Controller1 3715
EventTableActionAttach 16117: AttachmentParent=Tool_Arm_Pin_Right 3679, AttachmentChild=? -1, MountObject=false, Offset=[X=1, Y=0, Z=0, W=0, X=0, Y=1, Z=0, W=0, X=0, Y=0, Z=1, W=0, X=0, Y=0, Z=0, W=1], FlangeIndext=0, FindNearest=true
EventTableEntry 16118: Group=, Trigger=doAt_ArmP_Right 16119, Actions=[EventTableActionDetach 16120], Comment=, ActivationMode=2, Cyclic=false
EventTableTriggerIO 16119: IOValue=[0], IRC5Controller=? -1, Operator=0, SignalSource=Controller1 3715
EventTableActionDetach 16120: AttachmentParent=Tool_Arm_Pin_Right 3679, AttachmentChild=? -1
EventTableEntry 18691: Group=, Trigger=doGrepCaw 18692, Actions=[EventTableActionAttach 18693], Comment=, ActivationMode=2, Cyclic=false
EventTableTriggerIO 18692: IOValue=[1], IRC5Controller=? -1, Operator=0, SignalSource=Controller2 16804
EventTableActionAttach 18693: AttachmentParent=Tool_cow_catcher_Right 3685, AttachmentChild=? -1, MountObject=false, Offset=[X=1, Y=0, Z=0, W=0, X=0, Y=1, Z=0, W=0, X=0, Y=0, Z=1, W=0, X=0, Y=0, Z=0, W=1], FlangeIndext=0, FindNearest=true
EventTableEntry 18694: Group=, Trigger=doGrepCaw 18695, Actions=[EventTableActionDetach 18696], Comment=, ActivationMode=2, Cyclic=false
EventTableTriggerIO 18695: IOValue=[0], IRC5Controller=? -1, Operator=0, SignalSource=Controller2 16804
EventTableActionDetach 18696: AttachmentParent=Tool_cow_catcher_Right 3685, AttachmentChild=? -1
EventTableEntry 18697: Group=, Trigger=doGrepStak 18698, Actions=[EventTableActionAttach 18699], Comment=, ActivationMode=2, Cyclic=false
EventTableTriggerIO 18698: IOValue=[1], IRC5Controller=? -1, Operator=0, SignalSource=Controller2 16804
EventTableActionAttach 18699: AttachmentParent=Tool_Stack_Right 3670, AttachmentChild=? -1, MountObject=false, Offset=[X=1, Y=0, Z=0, W=0, X=0, Y=1, Z=0, W=0, X=0, Y=0, Z=1, W=0, X=0, Y=0, Z=0, W=1], FlangeIndext=0, FindNearest=true
EventTableEntry 18700: Group=, Trigger=doGrepStak 18701, Actions=[EventTableActionDetach 18702], Comment=, ActivationMode=2, Cyclic=false
EventTableTriggerIO 18701: IOValue=[0], IRC5Controller=? -1, Operator=0, SignalSource=Controller2 16804
EventTableActionDetach 18702: AttachmentParent=Tool_Stack_Right 3670, AttachmentChild=? -1
Station logic (signal -> signal, property => property):
  Controller1.diAttachTool -> SmartComponent_1.diAttachTool
  Controller1.doAttachTool -> SmartComponent_2.diAttachTool
  Controller1.doAttachTool -> SmartComponent_1.diAttachTool
  Controller1.doAttachTo_S -> SC_AttachTool_Right.diAttachTool
  Controller1.doAT_Left -> SC_AttachTool_left.diAT_Left
  Controller2.doAt_Tool_SC1 -> SmartComponent_1.di_Rob3_at_tool

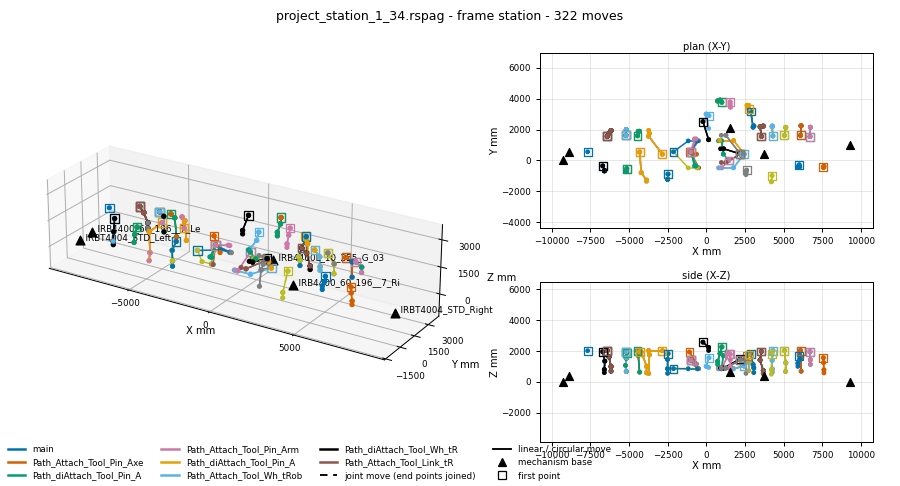
[picture p0: tool path of project_station_1_34.rspag in frame station, 322 of 322 moves have a stored position in this frame; points joined in program order, loops and branches not executed]
--- Backups/Controller1/RAPID/TASK1/PROGMOD/CalibData.mod ---
MODULE CalibData
    TASK PERS wobjdata InFeWOb_Lift_1:=[FALSE,TRUE,"",[[5841.89,-1164.97,60.5],[0.707107,0,0,-0.707107]],[[0,0,0],[1,0,0,0]]];
    TASK PERS wobjdata InFeWOb_Lift_2:=[FALSE,TRUE,"",[[4451.04,-1021.34,60.5],[0.707107,0,0,-0.707107]],[[0,0,0],[1,0,0,0]]];
    TASK PERS wobjdata InFeWOb_Lift_3:=[FALSE,TRUE,"",[[3089.54,-1164.97,60.5],[0.707107,0,0,-0.707107]],[[0,0,0],[1,0,0,0]]];
    TASK PERS wobjdata InFeWOb_Lift_4:=[FALSE,TRUE,"",[[1723.54,-1164.97,60.5],[0.707107,0,0,-0.707107]],[[0,0,0],[1,0,0,0]]];
    PERS tooldata Tool_Wheel:=[TRUE,[[0,0,380],[1,0,0,0]],[1,[0,0,1],[1,0,0,0],0,0,0]];
    PERS tooldata Tool_Link:=[TRUE,[[0,-15.353,170],[1,0,0,0]],[1,[0,0,1],[1,0,0,0],0,0,0]];
    PERS tooldata Tool_Stack:=[TRUE,[[0,50,519.006],[1,0,0,0]],[1,[0,0,1],[1,0,0,0],0,0,0]];
    PERS tooldata Tool_cow_catcher:=[TRUE,[[0,35.982,200],[1,0,0,0]],[1,[0,0,1],[1,0,0,0],0,0,0]];
    PERS tooldata Tool_Axelpin:=[TRUE,[[0,0,262.488],[1,0,0,0]],[1,[0,0,1],[1,0,0,0],0,0,0]];
    PERS tooldata Tool_ArmPin:=[TRUE,[[0,0,130.6],[1,0,0,0]],[1,[0,0,1],[1,0,0,0],0,0,0]];
    TASK PERS wobjdata TrLeFcWob:=[FALSE,TRUE,"",[[0,0,0],[1,0,0,0]],[[8517.76,-1485.75,283.772],[0.5,0.5,0.5,0.5]]];
    TASK PERS wobjdata stand_tool_Left:=[FALSE,TRUE,"",[[1478.6,679.135,195.515],[0.999999999,0,-0.000000533,-0.000035366]],[[0,0,0],[1,0,0,0]]];
ENDMODULE

--- Backups/Controller1/RAPID/TASK1/PROGMOD/Module1.mod ---
MODULE Module1
        CONST robtarget Target_10:=[[1201.24355653,0,1650],[0.5,0,0.866025404,0],[0,0,0,0],[0,9E+09,9E+09,9E+09,9E+09,9E+09]];
    CONST robtarget Target_20:=[[3963.854896054,-828.854630689,1454.480774594],[0.499999538,-0.000030628,0.86602567,0.000017683],[-1,0,-1,0],[4241.151152584,9E+09,9E+09,9E+09,9E+09,9E+09]];
    CONST robtarget Target_30:=[[2950.443314926,357.527946651,1454.481854801],[0.380191148,-0.562461624,0.658511194,0.32473777],[0,0,-1,0],[4241.151152584,9E+09,9E+09,9E+09,9E+09,9E+09]];
    CONST robtarget Target_40:=[[2995.943030468,644.935538293,1138.941403663],[0.290985601,-0.600036472,0.702502443,0.248543619],[0,0,-1,0],[4241.151152584,9E+09,9E+09,9E+09,9E+09,9E+09]];
    CONST robtarget Target_50:=[[3083.289734049,656.027413079,63.358505741],[0.000724262,-0.64994686,0.759956289,0.005915634],[0,0,-1,0],[4241.151152584,9E+09,9E+09,9E+09,9E+09,9E+09]];
    CONST robtarget Target_60:=[[4557.267950969,-828.812657397,1454.480142016],[0.499999538,-0.000030628,0.86602567,0.000017683],[-1,0,-1,0],[4834.564208984,9E+09,9E+09,9E+09,9E+09,9E+09]];
    CONST robtarget Target_70:=[[3666.847035703,331.436539168,1454.481091117],[0.396665539,-0.527226998,0.687045713,0.304395025],[0,0,-1,0],[4834.564208984,9E+09,9E+09,9E+09,9E+09,9E+09]];
    CONST robtarget Target_80:=[[3715.962548194,514.791066204,1187.071315354],[0.309979044,-0.56039355,0.730265947,0.237873302],[0,0,-1,0],[4834.564208984,9E+09,9E+09,9E+09,9E+09,9E+09]];
    CONST robtarget Target_90:=[[3672.961094398,706.430471729,-30.677697905],[0.007331935,-0.642677901,0.766101301,-0.000394066],[0,-1,-1,0],[4834.564208984,9E+09,9E+09,9E+09,9E+09,9E+09]];
    CONST robtarget Target_50_toFr:=[[3081.576625093,658.609917705,-196.623024223],[0.000724262,-0.64994686,0.759956289,0.005915634],[0,0,-1,0],[4241.151152584,9E+09,9E+09,9E+09,9E+09,9E+09]];
    CONST robtarget Target_100:=[[2203.019902359,391.487232107,1397.599561367],[0.177292135,-0.560008602,0.79971516,0.124151231],[0,0,-1,0],[3292.028188705,9E+09,9E+09,9E+09,9E+09,9E+09]];
    CONST robtarget Target_110:=[[2221.326956509,752.783157092,1010.114456714],[0.000865189,0.530640734,-0.847596301,-0.000415112],[0,0,0,0],[3292.028188705,9E+09,9E+09,9E+09,9E+09,9E+09]];
    CONST robtarget Target_120:=[[2221.326006337,752.783189439,110.114449536],[0.000865168,0.530640732,-0.847596303,-0.000415131],[0,0,0,0],[3292.028188705,9E+09,9E+09,9E+09,9E+09,9E+09]];

    CONST robtarget Target_130:=[[987.816935636,321.242307158,1454.483946964],[0,0.999999999,0.000035366,-0.000000533],[0,0,-1,0],[1865.816326531,9E+09,9E+09,9E+09,9E+09,9E+09]];
    CONST robtarget Target_140:=[[1103.153786786,521.044977306,1049.440867455],[0,0.999999999,0.000035366,-0.000000533],[0,-1,-1,0],[1865.816326531,9E+09,9E+09,9E+09,9E+09,9E+09]];
    CONST robtarget Target_150:=[[1236.539387975,687.447464624,430.260681798],[0,0.999999999,0.000035366,-0.000000533],[0,-1,-2,0],[1865.816326531,9E+09,9E+09,9E+09,9E+09,9E+09]];
    CONST robtarget Target_160:=[[1236.539068175,687.447464601,130.260681798],[0,0.999999999,0.000035366,-0.000000533],[0,-1,-2,0],[1865.816326531,9E+09,9E+09,9E+09,9E+09,9E+09]];

    CONST robtarget Target_170:=[[279.486006706,557.389955118,1399.5],[0.492935509,-0.145064645,0.853789347,0.083753111],[-1,0,-1,0],[6019.897959184,9E+09,9E+09,9E+09,9E+09,9E+09]];
    CONST robtarget Target_180:=[[618.789247384,530.377856509,1023.075191224],[0.35488033,-0.129929359,0.924494879,0.049875164],[-1,0,-1,0],[6264.246463776,9E+09,9E+09,9E+09,9E+09,9E+09]];
    CONST robtarget Target_190:=[[611.72,532.766550758,425],[0,0.241921897,0.970295726,0],[-1,0,0,0],[6264.246463776,9E+09,9E+09,9E+09,9E+09,9E+09]];
    CONST robtarget Target_Last:=[[611.72,532.766550758,125],[0,0.241921897,0.970295726,0],[-1,0,0,0],[6264.246463776,9E+09,9E+09,9E+09,9E+09,9E+09]];

!    CONST robtarget Target_200:=[[-71.078150076,641.700893198,1458.256],[0.482962913,-0.224143868,0.836516304,0.129409523],[-1,-1,0,0],[3054.32619099,9E+09,9E+09,9E+09,9E+09,9E+09]];
!    CONST robtarget Target_210:=[[120.387202333,608.657990735,1098.46641961],[0.374320881,-0.192085356,0.903690548,0.07956436],[-1,-1,0,0],[3054.32619099,9E+09,9E+09,9E+09,9E+09,9E+09]];
!    CONST robtarget Target_Ax_Last:=[[119.079,558.503550758,637.791],[0,0.707106781,0.707106781,0],[-1,0,1,0],[3054.32619099,9E+09,9E+09,9E+09,9E+09,9E+09]];

    CONST robtarget Target_200:=[[-71.078150076,641.700893198,1458.256],[0,0.999999999,0.000035366,-0.000000533],[-1,-1,-2,0],[3054.32619099,9E+09,9E+09,9E+09,9E+09,9E+09]];
    CONST robtarget Target_210:=[[120.387202333,608.657990735,1098.46641961],[0,0.999999999,0.000035366,-0.000000533],[-1,-1,-2,0],[3054.32619099,9E+09,9E+09,9E+09,9E+09,9E+09]];
    CONST robtarget Target_Ax_Last:=[[119.079,558.503550758,637.791],[0,0.999999999,0.000035366,-0.000000533],[-1,-1,-2,0],[3054.32619099,9E+09,9E+09,9E+09,9E+09,9E+09]];

    CONST robtarget Target_220:=[[-1005.987,117.427875173,1504.5],[0.183012702,-0.683012702,-0.683012702,-0.183012702],[0,-1,0,0],[3220,9E+09,9E+09,9E+09,9E+09,9E+09]];
    CONST robtarget Target_230_2:=[[812.378542163,565.582550758,584.485],[0,0.707106781,0.707106781,0],[-1,0,1,0],[4718.142857143,9E+09,9E+09,9E+09,9E+09,9E+09]];
    CONST robtarget Target_Link_lqa:=[[880.315,555.582550758,159.485],[0,0.707106781,0.707106781,0],[-1,0,1,0],[4718.142857143,9E+09,9E+09,9E+09,9E+09,9E+09]];
    CONST robtarget Target_230:=[[327.127875173,215.749857143,1504.5],[0,0.707106781,0.707106781,0],[-1,-1,0,0],[4682.142857143,9E+09,9E+09,9E+09,9E+09,9E+09]];
    CONST robtarget Target_240:=[[812.378542163,565.582550758,584.485],[0,0.707106781,0.707106781,0],[-1,0,1,0],[4718.142857143,9E+09,9E+09,9E+09,9E+09,9E+09]];
    CONST robtarget Target_250:=[[-251.948219969,453.119934775,1524.2],[0.460252427,-0.338383084,0.797180587,0.195365564],[-1,-1,0,0],[907.571211037,9E+09,9E+09,9E+09,9E+09,9E+09]];
    CONST robtarget Target_260:=[[46.568796881,586.853509114,912.209220086],[0.170740423,-0.179466959,0.968317056,0.031644867],[-1,-1,0,0],[1361.357430131,9E+09,9E+09,9E+09,9E+09,9E+09]];
    CONST robtarget Target_270:=[[69.179,556.469550758,371.21242788],[0.017451742,-0.008251102,0.999809624,0.002841082],[-1,-1,0,0],[1361.357430131,9E+09,9E+09,9E+09,9E+09,9E+09]];
    CONST robtarget Target_ArmPin_Last:=[[69.179,556.469550758,171.21242788],[0.017451742,-0.008251102,0.999809624,0.002841082],[-1,-1,0,0],[1361.357430131,9E+09,9E+09,9E+09,9E+09,9E+09]];
    CONST robtarget Target_280:=[[1485.75,761.336341228,-649.921518108],[0.703968023,0.0665509,0.0665509,-0.703968023],[0,-1,0,0],[6533.480857081,9E+09,9E+09,9E+09,9E+09,9E+09]];
    CONST robtarget Target_290:=[[1470.397,1281.228,-726.945186051],[0.683012702,0.183012702,0.183012702,-0.683012702],[-1,0,-1,0],[6442.346938776,9E+09,9E+09,9E+09,9E+09,9E+09]];
    CONST robtarget Target_300:=[[2196.413,199.691,-132.387449242],[0.707106781,0,0,-0.707106781],[0,0,-1,0],[6900,9E+09,9E+09,9E+09,9E+09,9E+09]];
    CONST robtarget Target_Wheel_Left_B:=[[450.735,199.691,-132.387449242],[1,0,0,0],[-1,-1,1,0],[6900,9E+09,9E+09,9E+09,9E+09,9E+09]];
    CONST robtarget Target_Wheel_Left_F:=[[2196.413,199.691,-132.387449242],[1,0,0,0],[0,0,0,0],[6900,9E+09,9E+09,9E+09,9E+09,9E+09]];
    CONST robtarget Target_AxelPin_Left_B:=[[446.737,199.434,-208.902449242],[0.707106781,0,0,-0.707106781],[-1,-1,0,0],[6760.374761202,9E+09,9E+09,9E+09,9E+09,9E+09]];
    CONST robtarget Target_AxelPin_Left_F:=[[2192.848,199.434,-209.134449242],[0.707106781,0,0,-0.707106781],[0,0,-1,0],[6533.480857081,9E+09,9E+09,9E+09,9E+09,9E+09]];
    CONST robtarget Target_Link_Left:=[[1327.179,502.16,-268.354449242],[0.707106781,0,0,-0.707106781],[-1,1,-2,0],[6533.480857081,9E+09,9E+09,9E+09,9E+09,9E+09]];
    CONST robtarget Target_ArmPin_Left_B:=[[575.179,512.16,-308.354449242],[0.707106781,0,0,-0.707106781],[-1,-1,0,0],[6533.479789407,9E+09,9E+09,9E+09,9E+09,9E+09]];
    CONST robtarget Target_ArmPin_Left_F:=[[2325.179,512.16,-308.354449242],[0.707106781,0,0,-0.707106781],[0,0,-1,0],[6533.479789407,9E+09,9E+09,9E+09,9E+09,9E+09]];
    CONST robtarget Target_Pre_AxelPin_Left:=[[1485.75,207.778427238,-1763.832931776],[0.707106625,-0.000469668,-0.000469668,-0.707106625],[0,0,0,0],[4852.213289649,9E+09,9E+09,9E+09,9E+09,9E+09]];
    CONST robtarget Target_Wheel_Left_Pre_B:=[[450.735,199.691,-232.387449242],[1,0,0,0],[-1,-1,1,0],[6900,9E+09,9E+09,9E+09,9E+09,9E+09]];
    CONST robtarget Target_Wheel_Left_Pre_F:=[[2196.413,199.691,-232.387449242],[1,0,0,0],[0,0,0,0],[6900,9E+09,9E+09,9E+09,9E+09,9E+09]];
    CONST robtarget Target_AxelPin_Left_Pre_B:=[[446.737,199.434,-808.902449242],[0.707106781,0,0,-0.707106781],[-1,-1,0,0],[6760.374761202,9E+09,9E+09,9E+09,9E+09,9E+09]];
    CONST robtarget Target_AxelPin_Left_Pre:=[[1485.75,207.778427238,-1763.832931776],[0.707106625,-0.000469668,-0.000469668,-0.707106625],[0,0,0,0],[4852.213289649,9E+09,9E+09,9E+09,9E+09,9E+09]];
    CONST robtarget Target_AxelPin_Left_Pre_F:=[[2192.848,199.434,-809.134449242],[0.707106781,0,0,-0.707106781],[0,0,-1,0],[6533.480857081,9E+09,9E+09,9E+09,9E+09,9E+09]];
    CONST robtarget Target_Link_Left_Pre:=[[1470.397,1281.228,-726.945186051],[0.683012702,0.183012702,0.183012702,-0.683012702],[-1,0,-1,0],[6442.346938776,9E+09,9E+09,9E+09,9E+09,9E+09]];
    CONST robtarget Target_ArmPin_Left_Pre_B:=[[575.179,512.16,-408.354449242],[0.707106781,0,0,-0.707106781],[-1,-1,0,0],[6533.479789407,9E+09,9E+09,9E+09,9E+09,9E+09]];
    CONST robtarget Target_ArmPin_Left_Pre:=[[1485.75,761.336341228,-649.921518108],[0.703968023,0.0665509,0.0665509,-0.703968023],[0,-1,0,0],[6533.480857081,9E+09,9E+09,9E+09,9E+09,9E+09]];
    CONST robtarget Target_ArmPin_Left_Pre_F:=[[2325.179,512.16,-408.354449242],[0.707106781,0,0,-0.707106781],[0,0,-1,0],[6533.479789407,9E+09,9E+09,9E+09,9E+09,9E+09]];
!***********************************************************
    !
    ! Module:  Module1
    !
    ! Description:
    !   <Insert description here>
    !
    ! Author: haba0028
    !
    ! Version: 1.0
    !
    !***********************************************************


    !***********************************************************
    !
    ! Procedure main
    !
    !   This is the entry point of your program
    !
    !***********************************************************
    PROC main()
        !Add your code here
        SetDO doAttachTool,0;
        SetDO doAT_Left,0;

        SetDO doAt_Wh_Left,0;
        SetDO doAt_Link_Left,0;
        SetDO doAt_AxelP_Left,0;
        SetDO doAt_Arm_Left,0;



!        Path_Attach_Tool_Wh_tRob_Left;
!        Path_At_Wh_tR_Left;
!        Path_diAt_Wh_tR_Left;
!        Path_diAttach_Wh_tRob_Left;


!        Path_Attach_Tool_Pin_Axel;
!        Path_At_AxP_tR_Left;
!        Path_At_diAxP_tR_Left;
!        Path_diAttach_Tool_Pin_Axel;



!        Path_Attach_Link_tRob_Left;
!        Path_At_Link_tR_Left;
!        Path_diAt_Link_tR_Left;
!        Path_diAttach_Link_tRob_Left;


!        Path_Attach_Tool_Pin_Arm;
!        Path_At_ArP_tR_Left;
!        Path_diAt_ArP_tR_Left;
!        Path_diAttach_Tool_Pin_Arm;

!!!!!

        Path_Attach_Tool_Wh_tRob_Left;
        Path_At_Wh_tR_Left;
        Path_At_WtT_Left_B;
        Path_At_Wh_tR_Left;
        Path_At_WtT_Left_F;
        Path_diAttach_Tool_Wh_tRob_Left;

        Path_Attach_Tool_Pin_Axel;
        Path_At_AxP_tR_Left;
        Path_At_AxPT_Left_B;
        Path_At_AxP_tR_Left;
        Path_At_AxPT_Left_F;
        Path_diAttach_Tool_Pin_Axel;


         Path_Attach_Tool_Link_tRob_Left;
         Path_At_Link_tR_Left;
         Path_At_Link_tT_Left;
         Path_diAttach_Tool_Link_tRo_Left;

         Path_Attach_Tool_Pin_Arm;
         Path_At_ArP_tR_Left;
         Path_At_ArP_tT_Left_B;
         Path_At_ArP_tR_Left;
         Path_At_ArP_tT_Left_F;
         Path_diAttach_Tool_Pin_Arm;

         MoveJ Target_10,v1000,fine,tool0\WObj:=wobj0;  ! Move To Home
         !!!
    ENDPROC



    PROC Path_Attach_Tool_Pin_Axel()
!        MoveL Target_10,v1000,fine,tool0\WObj:=wobj0;
!        MoveL Target_20,v1000,fine,tool0\WObj:=stand_tool_Left;
        MoveJ Target_30,v1000,fine,tool0\WObj:=stand_tool_Left;
        MoveL Target_40,v1000,fine,tool0\WObj:=stand_tool_Left;
        MoveL Target_50,v1000,fine,tool0\WObj:=stand_tool_Left;
        WaitTime 0.4;
!        SetDO doAttachTool,1;
        SetDO doAT_Left,1;
        WaitTime 1;
        MoveL Target_40,v1000,fine,Tool_Axelpin\WObj:=stand_tool_Left;
        MoveL Target_30,v1000,fine,Tool_Axelpin\WObj:=stand_tool_Left;
!        MoveL Target_20,v1000,fine,Tool_Axelpin\WObj:=stand_tool_Left;
    ENDPROC

    PROC Path_diAttach_Tool_Pin_Axel()
        !MoveL Target_10,v1000,fine,tool0\WObj:=wobj0;
!        MoveL Target_20,v1000,fine,Tool_Axelpin\WObj:=stand_tool_Left;
        MoveJ Target_30,v1000,fine,Tool_Axelpin\WObj:=stand_tool_Left;
        MoveL Target_40,v1000,fine,Tool_Axelpin\WObj:=stand_tool_Left;
        MoveL Target_50,v1000,fine,tool0\WObj:=stand_tool_Left;
        WaitTime 0.4;
!        SetDO doAttachTool,0;
        SetDO doAT_Left,0;
        WaitTime 1;
        MoveL Target_40,v1000,fine,tool0\WObj:=stand_tool_Left;
        MoveL Target_30,v1000,fine,tool0\WObj:=stand_tool_Left;
!        MoveL Target_20,v1000,fine,tool0\WObj:=stand_tool_Left;
    ENDPROC



    PROC Path_Attach_Tool_Pin_Arm()
!        MoveJ Target_10,v1000,fine,tool0\WObj:=wobj0;
        MoveJ Target_60,v1000,fine,tool0\WObj:=stand_tool_Left;
        MoveL Target_70,v1000,fine,tool0\WObj:=stand_tool_Left;
        MoveL Target_80,v1000,fine,tool0\WObj:=stand_tool_Left;
        MoveL Target_90,v1000,fine,tool0\WObj:=stand_tool_Left;
        WaitTime 0.4;
        SetDO doAT_Left,1;
        WaitTime 1;
        MoveL Target_80,v1000,fine,Tool_ArmPin\WObj:=stand_tool_Left;
        MoveL Target_70,v1000,fine,Tool_ArmPin\WObj:=stand_tool_Left;
        MoveL Target_60,v1000,fine,Tool_ArmPin\WObj:=stand_tool_Left;
    ENDPROC

    PROC Path_diAttach_Tool_Pin_Arm()
        !MoveL Target_10,v1000,fine,tool0\WObj:=wobj0;
        MoveJ Target_60,v1000,fine,Tool_ArmPin\WObj:=stand_tool_Left;
        MoveL Target_70,v1000,fine,Tool_ArmPin\WObj:=stand_tool_Left;
        MoveL Target_80,v1000,fine,Tool_ArmPin\WObj:=stand_tool_Left;
        MoveL Target_90,v1000,fine,tool0\WObj:=stand_tool_Left;
        WaitTime 0.4;
        SetDO doAT_Left,0;
        WaitTime 1;
        MoveL Target_80,v1000,fine,tool0\WObj:=stand_tool_Left;
        MoveL Target_70,v1000,fine,tool0\WObj:=stand_tool_Left;
        MoveL Target_60,v1000,fine,tool0\WObj:=stand_tool_Left;
    ENDPROC



    PROC Path_Attach_Tool_Wh_tRob_Left()
        WaitTime 0.3;
        MoveJ Target_100,v1000,fine,tool0\WObj:=stand_tool_Left;
        MoveL Target_110,v1000,fine,tool0\WObj:=stand_tool_Left;
        MoveL Target_120,v1000,fine,tool0\WObj:=stand_tool_Left;
        WaitTime 0.4;
        SetDO doAT_Left,1;
        WaitTime 1;
        MoveL Target_110,v1000,fine,Tool_Wheel\WObj:=stand_tool_Left;
        MoveL Target_100,v1000,fine,Tool_Wheel\WObj:=stand_tool_Left;
    ENDPROC
    PROC Path_diAttach_Tool_Wh_tRob_Left()
        WaitTime 0.3;
        MoveJ Target_100,v1000,fine,Tool_Wheel\WObj:=stand_tool_Left;
        MoveL Target_110,v1000,fine,Tool_Wheel\WObj:=stand_tool_Left;
        MoveL Target_120,v1000,fine,tool0\WObj:=stand_tool_Left;
        WaitTime 0.4;
        SetDO doAT_Left,0;
        WaitTime 1;
        MoveL Target_110,v1000,fine,tool0\WObj:=stand_tool_Left;
        MoveL Target_100,v1000,fine,tool0\WObj:=stand_tool_Left;
    ENDPROC


    PROC Path_Attach_Tool_Link_tRob_Left()
        WaitTime 0.4;
        MoveJ Target_130,v1000,fine,tool0\WObj:=stand_tool_Left;
        MoveL Target_140,v1000,fine,tool0\WObj:=stand_tool_Left;
        MoveL Target_150,v1000,fine,tool0\WObj:=stand_tool_Left;
        MoveL Target_160,v1000,fine,tool0\WObj:=stand_tool_Left;
        WaitTime 0.4;
        SetDO doAT_Left,1;
        WaitTime 1;
        MoveL Target_150,v1000,fine,Tool_Link\WObj:=stand_tool_Left;
        MoveL Target_140,v1000,fine,Tool_Link\WObj:=stand_tool_Left;
        MoveL Target_130,v1000,fine,Tool_Link\WObj:=stand_tool_Left;
    ENDPROC
    PROC Path_diAttach_Tool_Link_tRo_Left()
        WaitTime 0.4;
        MoveJ Target_130,v1000,fine,Tool_Link\WObj:=stand_tool_Left;
        MoveL Target_140,v1000,fine,Tool_Link\WObj:=stand_tool_Left;
        MoveL Target_150,v1000,fine,Tool_Link\WObj:=stand_tool_Left;
        MoveL Target_160,v1000,fine,tool0\WObj:=stand_tool_Left;
        WaitTime 0.4;
        SetDO doAT_Left,0;
        WaitTime 1;
        MoveL Target_150,v1000,fine,tool0\WObj:=stand_tool_Left;
        MoveL Target_140,v1000,fine,tool0\WObj:=stand_tool_Left;
        MoveL Target_130,v1000,fine,tool0\WObj:=stand_tool_Left;
    ENDPROC


    PROC Path_At_Wh_tR_Left()
        WaitTime 0.4;
        MoveJ Target_170,v1000,fine,Tool_Wheel\WObj:=InFeWOb_Lift_1;
        MoveL Target_180,v1000,fine,Tool_Wheel\WObj:=InFeWOb_Lift_1;
        MoveL Target_190,v1000,fine,Tool_Wheel\WObj:=InFeWOb_Lift_1;
        MoveL Target_Last,v1000,fine,Tool_Wheel\WObj:=InFeWOb_Lift_1;
        WaitTime 0.4;
!        SetDO doAT_Left,1;
        SetDO doAt_Wh_Left,1;
        WaitTime 1;
        MoveL Target_190,v1000,fine,Tool_Wheel\WObj:=InFeWOb_Lift_1;
        MoveL Target_180,v1000,fine,Tool_Wheel\WObj:=InFeWOb_Lift_1;
        MoveL Target_170,v1000,fine,Tool_Wheel\WObj:=InFeWOb_Lift_1;
    ENDPROC
    PROC Path_diAt_Wh_tR_Left()
        WaitTime 0.4;
        MoveJ Target_170,v1000,fine,Tool_Wheel\WObj:=InFeWOb_Lift_1;
        MoveL Target_180,v1000,fine,Tool_Wheel\WObj:=InFeWOb_Lift_1;
        MoveL Target_190,v1000,fine,Tool_Wheel\WObj:=InFeWOb_Lift_1;
        MoveL Target_Last,v1000,fine,Tool_Wheel\WObj:=InFeWOb_Lift_1;
        WaitTime 0.4;
!        SetDO doAT_Left,0;
        SetDO doAt_Wh_Left,0;
        WaitTime 1;
        MoveL Target_190,v1000,fine,Tool_Wheel\WObj:=InFeWOb_Lift_1;
        MoveL Target_180,v1000,fine,Tool_Wheel\WObj:=InFeWOb_Lift_1;
        MoveL Target_170,v1000,fine,Tool_Wheel\WObj:=InFeWOb_Lift_1;
    ENDPROC

    PROC Path_At_AxP_tR_Left()
        WaitTime 0.4;
        MoveJ Target_200,v1000,fine,Tool_Axelpin\WObj:=InFeWOb_Lift_3;
        MoveL Target_210,v1000,fine,Tool_Axelpin\WObj:=InFeWOb_Lift_3;
        MoveL Target_Ax_Last,v1000,fine,Tool_Axelpin\WObj:=InFeWOb_Lift_3;
        WaitTime 0.4;
        SetDO doAt_AxelP_Left,1;
        WaitTime 1;
        MoveL Target_210,v1000,fine,Tool_Axelpin\WObj:=InFeWOb_Lift_3;
        MoveL Target_200,v1000,fine,Tool_Axelpin\WObj:=InFeWOb_Lift_3;
    ENDPROC
    PROC Path_At_diAxP_tR_Left()
        WaitTime 0.4;
        MoveJ Target_200,v1000,fine,Tool_Axelpin\WObj:=InFeWOb_Lift_3;
        MoveL Target_210,v1000,fine,Tool_Axelpin\WObj:=InFeWOb_Lift_3;
        MoveL Target_Ax_Last,v1000,fine,Tool_Axelpin\WObj:=InFeWOb_Lift_3;
        WaitTime 0.4;
        SetDO doAt_AxelP_Left,0;
        WaitTime 1;
        MoveL Target_210,v1000,fine,Tool_Axelpin\WObj:=InFeWOb_Lift_3;
        MoveL Target_200,v1000,fine,Tool_Axelpin\WObj:=InFeWOb_Lift_3;
    ENDPROC

    PROC Path_At_Link_tR_Left()
        WaitTime 0.4;
        MoveJ Target_220,v1000,fine,Tool_Link\WObj:=InFeWOb_Lift_2;
        MoveL Target_230,v1000,fine,Tool_Link\WObj:=InFeWOb_Lift_2;
        MoveL Target_240,v1000,fine,Tool_Link\WObj:=InFeWOb_Lift_2;
        MoveL Target_Link_lqa,v1000,fine,Tool_Link\WObj:=InFeWOb_Lift_2;
        WaitTime 0.4;
        SetDO doAt_Link_Left,1;
        WaitTime 1;
        MoveL Target_240,v1000,fine,Tool_Link\WObj:=InFeWOb_Lift_2;
        MoveL Target_230,v1000,fine,Tool_Link\WObj:=InFeWOb_Lift_2;
        MoveL Target_220,v1000,fine,Tool_Link\WObj:=InFeWOb_Lift_2;
    ENDPROC
    PROC Path_diAt_Link_tR_Left()
        WaitTime 0.4;
        MoveJ Target_220,v1000,fine,Tool_Link\WObj:=InFeWOb_Lift_2;
        MoveL Target_230,v1000,fine,Tool_Link\WObj:=InFeWOb_Lift_2;
        MoveL Target_240,v1000,fine,Tool_Link\WObj:=InFeWOb_Lift_2;
        MoveL Target_Link_lqa,v1000,fine,Tool_Link\WObj:=InFeWOb_Lift_2;
        WaitTime 0.4;
        SetDO doAt_Link_Left,0;
        WaitTime 1;
        MoveL Target_240,v1000,fine,Tool_Link\WObj:=InFeWOb_Lift_2;
        MoveL Target_230,v1000,fine,Tool_Link\WObj:=InFeWOb_Lift_2;
        MoveL Target_220,v1000,fine,Tool_Link\WObj:=InFeWOb_Lift_2;
    ENDPROC

    PROC Path_At_ArP_tR_Left()
        WaitTime 0.4;
        MoveJ Target_250,v1000,fine,Tool_ArmPin\WObj:=InFeWOb_Lift_4;
        MoveL Target_260,v1000,fine,Tool_ArmPin\WObj:=InFeWOb_Lift_4;
        MoveL Target_270,v1000,fine,Tool_ArmPin\WObj:=InFeWOb_Lift_4;
        MoveL Target_ArmPin_Last,v1000,fine,Tool_ArmPin\WObj:=InFeWOb_Lift_4;
        WaitTime 0.4;
        SetDO doAt_Arm_Left,1;
        WaitTime 1;
        MoveL Target_270,v1000,fine,Tool_ArmPin\WObj:=InFeWOb_Lift_4;
        MoveL Target_260,v1000,fine,Tool_ArmPin\WObj:=InFeWOb_Lift_4;
        MoveL Target_250,v1000,fine,Tool_ArmPin\WObj:=InFeWOb_Lift_4;
    ENDPROC
    PROC Path_diAt_ArP_tR_Left()
        WaitTime 0.4;
        MoveJ Target_250,v1000,fine,Tool_ArmPin\WObj:=InFeWOb_Lift_4;
        MoveL Target_260,v1000,fine,Tool_ArmPin\WObj:=InFeWOb_Lift_4;
        MoveL Target_270,v1000,fine,Tool_ArmPin\WObj:=InFeWOb_Lift_4;
        MoveL Target_ArmPin_Last,v1000,fine,Tool_ArmPin\WObj:=InFeWOb_Lift_4;
        WaitTime 0.4;
        SetDO doAt_Arm_Left,0;
        WaitTime 1;
        MoveL Target_270,v1000,fine,Tool_ArmPin\WObj:=InFeWOb_Lift_4;
        MoveL Target_260,v1000,fine,Tool_ArmPin\WObj:=InFeWOb_Lift_4;
        MoveL Target_250,v1000,fine,Tool_ArmPin\WObj:=InFeWOb_Lift_4;
    ENDPROC

    PROC Path_At_WtT_Left_B()
        WaitTime 0.4;
        MoveJ Target_280,v1000,fine,Tool_Wheel\WObj:=TrLeFcWob;
        MoveL Target_Wheel_Left_Pre_B,v1000,fine,Tool_Axelpin\WObj:=TrLeFcWob;
        MoveL Target_Wheel_Left_B,v1000,fine,Tool_Wheel\WObj:=TrLeFcWob;
        WaitTime 0.4;
        SetDO doAt_Wh_Left,0;
        WaitTime 1;
        MoveL Target_280,v1000,fine,Tool_Wheel\WObj:=TrLeFcWob;
    ENDPROC
    PROC Path_AT_WtT_Left_F()
        WaitTime 0.4;
        MoveJ Target_280,v1000,fine,Tool_Wheel\WObj:=TrLeFcWob;
        MoveL Target_Wheel_Left_Pre_F,v1000,fine,Tool_Axelpin\WObj:=TrLeFcWob;
        MoveL Target_Wheel_Left_F,v1000,fine,Tool_Wheel\WObj:=TrLeFcWob;
        WaitTime 0.4;
        SetDO doAt_Wh_Left,0;
        WaitTime 1;
        MoveL Target_280,v1000,fine,Tool_Wheel\WObj:=TrLeFcWob;
    ENDPROC

    PROC Path_At_AxPT_Left_B()
        WaitTime 0.4;
        MoveJ Target_AxelPin_Left_Pre,v1000,fine,Tool_Axelpin\WObj:=TrLeFcWob;
        MoveL Target_AxelPin_Left_Pre_B,v1000,fine,Tool_Axelpin\WObj:=TrLeFcWob;
        MoveL Target_AxelPin_Left_B,v1000,fine,Tool_Axelpin\WObj:=TrLeFcWob;
        WaitTime 0.4;
        SetDO doAt_AxelP_Left,0;
        WaitTime 1;
        MoveL Target_280,v1000,fine,Tool_Axelpin\WObj:=TrLeFcWob;
    ENDPROC
    PROC Path_At_AxPT_Left_F()
        WaitTime 0.4;
        MoveJ Target_AxelPin_Left_Pre,v1000,fine,Tool_Axelpin\WObj:=TrLeFcWob;
        MoveL Target_AxelPin_Left_Pre_F,v1000,fine,Tool_Axelpin\WObj:=TrLeFcWob;
        MoveL Target_AxelPin_Left_F,v1000,fine,Tool_Axelpin\WObj:=TrLeFcWob;
        WaitTime 0.4;
        SetDO doAt_AxelP_Left,0;
        WaitTime 1;
        MoveL Target_280,v1000,fine,Tool_Axelpin\WObj:=TrLeFcWob;
    ENDPROC


    PROC Path_At_Link_tT_Left()
        WaitTime 0.4;
        MoveJ Target_Link_Left_Pre,v1000,fine,Tool_Link\WObj:=TrLeFcWob;
        MoveL Target_Link_Left,v1000,fine,Tool_Link\WObj:=TrLeFcWob;
        WaitTime 0.4;
        SetDO doAt_Link_Left,0;
        WaitTime 1;
        MoveL Target_Link_Left_Pre,v1000,fine,Tool_Link\WObj:=TrLeFcWob;
    ENDPROC

    PROC Path_At_ArP_tT_Left_B()
        WaitTime 0.4;
        MoveJ Target_ArmPin_Left_Pre,v1000,fine,Tool_Axelpin\WObj:=TrLeFcWob;
        MoveL Target_ArmPin_Left_Pre_B,v1000,fine,Tool_Axelpin\WObj:=TrLeFcWob;
        MoveL Target_ArmPin_Left_B,v1000,fine,Tool_ArmPin\WObj:=TrLeFcWob;
        WaitTime 0.4;
        SetDO doAt_Arm_Left,0;
        WaitTime 1;
        MoveL Target_ArmPin_Left_Pre,v1000,fine,Tool_Axelpin\WObj:=TrLeFcWob;
    ENDPROC
    PROC Path_At_ArP_tT_Left_F()
        WaitTime 0.4;
        MoveJ Target_ArmPin_Left_Pre,v1000,fine,Tool_Axelpin\WObj:=TrLeFcWob;
        MoveL Target_ArmPin_Left_Pre_F,v1000,fine,Tool_Axelpin\WObj:=TrLeFcWob;
        MoveL Target_ArmPin_Left_F,v1000,fine,Tool_ArmPin\WObj:=TrLeFcWob;
        WaitTime 0.4;
        SetDO doAt_Arm_Left,0;
        WaitTime 1;
        MoveL Target_ArmPin_Left_Pre,v1000,fine,Tool_Axelpin\WObj:=TrLeFcWob;
    ENDPROC
    PROC Path_Attach_Wh_tRob_Left()
        WaitTime 0.3;
        MoveJ Target_100,v1000,fine,tool0\WObj:=stand_tool_Left;
        MoveL Target_110,v1000,fine,tool0\WObj:=stand_tool_Left;
        MoveL Target_120,v1000,fine,tool0\WObj:=stand_tool_Left;
        WaitTime 0.4;
        SetDO doAT_Left,1;
        WaitTime 1;
        MoveL Target_110,v1000,fine,Tool_Wheel\WObj:=stand_tool_Left;
        MoveL Target_100,v1000,fine,Tool_Wheel\WObj:=stand_tool_Left;
    ENDPROC
    PROC Path_diAttach_Wh_tRob_Left()
        WaitTime 0.3;
        MoveJ Target_100,v1000,fine,Tool_Wheel\WObj:=stand_tool_Left;
        MoveL Target_110,v1000,fine,Tool_Wheel\WObj:=stand_tool_Left;
        MoveL Target_120,v1000,fine,tool0\WObj:=stand_tool_Left;
        WaitTime 0.4;
        SetDO doAT_Left,0;
        WaitTime 1;
        MoveL Target_110,v1000,fine,tool0\WObj:=stand_tool_Left;
        MoveL Target_100,v1000,fine,tool0\WObj:=stand_tool_Left;
    ENDPROC
    PROC Path_Attach_Link_tRob_Left()
        WaitTime 0.4;
        MoveL Target_130,v1000,fine,tool0\WObj:=stand_tool_Left;
        MoveL Target_140,v1000,fine,tool0\WObj:=stand_tool_Left;
        MoveL Target_150,v1000,fine,tool0\WObj:=stand_tool_Left;
        MoveL Target_160,v1000,fine,tool0\WObj:=stand_tool_Left;
        WaitTime 0.4;
        SetDO doAT_Left,1;
        WaitTime 1;
        MoveL Target_150,v1000,fine,Tool_Link\WObj:=stand_tool_Left;
        MoveL Target_140,v1000,fine,Tool_Link\WObj:=stand_tool_Left;
        MoveL Target_130,v1000,fine,Tool_Link\WObj:=stand_tool_Left;
    ENDPROC
    PROC Path_diAttach_Link_tRob_Left()
        WaitTime 0.4;
        MoveL Target_130,v1000,fine,Tool_Link\WObj:=stand_tool_Left;
        MoveL Target_140,v1000,fine,Tool_Link\WObj:=stand_tool_Left;
        MoveL Target_150,v1000,fine,Tool_Link\WObj:=stand_tool_Left;
        MoveL Target_160,v1000,fine,tool0\WObj:=stand_tool_Left;
        WaitTime 0.4;
        SetDO doAT_Left,0;
        WaitTime 1;
        MoveL Target_150,v1000,fine,tool0\WObj:=stand_tool_Left;
        MoveL Target_140,v1000,fine,tool0\WObj:=stand_tool_Left;
        MoveL Target_130,v1000,fine,tool0\WObj:=stand_tool_Left;
    ENDPROC

ENDMODULE

--- Backups/Controller1/RAPID/TASK2/PROGMOD/CalibData.mod ---
MODULE CalibData

    TASK PERS wobjdata stand_tool_2:=[FALSE,TRUE,"",[[16226.9,2322.72,195.515],[0.000035473,0.000000533,0,0.999999999]],[[0,0,0],[1,0,0,0]]];
    TASK PERS wobjdata InFeWOb_Right_1:=[FALSE,TRUE,"",[[10894.2,-864.97,60.5],[0.707107,0,0,-0.707107]],[[0,0,0],[1,0,0,0]]];
    TASK PERS wobjdata InFeWOb_Right_2:=[FALSE,TRUE,"",[[12560.2,-864.97,60.5],[0.707107,0,0,-0.707107]],[[0,0,0],[1,0,0,0]]];
    TASK PERS wobjdata InFeWOb_Right_3:=[FALSE,TRUE,"",[[14226.2,-864.97,60.5],[0.707107,0,0,-0.707107]],[[0,0,0],[1,0,0,0]]];
    TASK PERS wobjdata InFeWOb_Right_4:=[FALSE,TRUE,"",[[15892.2,-864.97,60.5],[0.707107,0,0,-0.707107]],[[0,0,0],[1,0,0,0]]];
    PERS tooldata Tool_Wheel:=[TRUE,[[0,0,380],[1,0,0,0]],[1,[0,0,1],[1,0,0,0],0,0,0]];
    PERS tooldata Tool_Link:=[TRUE,[[0,-15.353,170],[1,0,0,0]],[1,[0,0,1],[1,0,0,0],0,0,0]];
    PERS tooldata Tool_Stack:=[TRUE,[[0,50,519.006],[1,0,0,0]],[1,[0,0,1],[1,0,0,0],0,0,0]];
    PERS tooldata Tool_cow_catcher:=[TRUE,[[0,35.982,200],[1,0,0,0]],[1,[0,0,1],[1,0,0,0],0,0,0]];
    PERS tooldata Tool_Axelpin:=[TRUE,[[0,0,262.488],[1,0,0,0]],[1,[0,0,1],[1,0,0,0],0,0,0]];
    PERS tooldata Tool_ArmPin:=[TRUE,[[0,0,130.6],[1,0,0,0]],[1,[0,0,1],[1,0,0,0],0,0,0]];
    TASK PERS wobjdata TrRiFcWOb:=[FALSE,TRUE,"",[[0,558.721,0],[1,0,0,0]],[[9517.76,-2044.47,283.772],[0.5,0.5,0.5,0.5]]];
    TASK PERS wobjdata stand_tool_Right:=[FALSE,TRUE,"",[[16226.9,2322.72,195.515],[0.000035473,0.000000533,0,0.999999999]],[[0,0,0],[1,0,0,0]]];
ENDMODULE

--- Backups/Controller1/RAPID/TASK2/PROGMOD/Module1.mod ---
MODULE Module1
        CONST robtarget Target_50:=[[16593.174986227,-138.169431595,1650],[0,0.866025404,0,-0.5],[0,-1,0,0],[0,9E+09,9E+09,9E+09,9E+09,9E+09]];
    CONST robtarget Target_40:=[[1760.356554662,2461.009343776,1390.33688758],[0.14458959,-0.000035188,0.989491713,0.000005141],[-1,0,-1,0],[2208,9E+09,9E+09,9E+09,9E+09,9E+09]];
    CONST robtarget Target_30:=[[640.377241487,1340.870083489,1390.338081562],[0.102243944,0.69965099,0.699701501,-0.10223736],[-2,0,-1,0],[2208,9E+09,9E+09,9E+09,9E+09,9E+09]];
    CONST robtarget Target_20:=[[620.419562878,735.592491307,865.144352753],[0.006170459,0.707054502,0.70710521,-0.006170772],[-2,0,-1,0],[2208,9E+09,9E+09,9E+09,9E+09,9E+09]];
    CONST robtarget Target_10:=[[620.419245661,735.592627753,567.78600829],[0.006170449,0.707054533,0.707105179,-0.006170762],[-2,0,-1,0],[2208,9E+09,9E+09,9E+09,9E+09,9E+09]];
    CONST robtarget Target_60:=[[2209.55196843,2461.046196662,1454.482644432],[0.499999538,-0.000030721,0.86602567,0.000017736],[-1,0,-1,0],[2576,9E+09,9E+09,9E+09,9E+09,9E+09]];
    CONST robtarget Target_70:=[[1248.946636989,1259.734486003,1454.483668529],[0.353565606,0.612350524,0.612394346,-0.353541175],[-1,-1,0,0],[2576,9E+09,9E+09,9E+09,9E+09,9E+09]];
    CONST robtarget Target_80:=[[1226.845337589,640.610759838,978.085457621],[0.122791813,0.696339217,0.696389262,-0.122783798],[-1,-1,0,0],[2576,9E+09,9E+09,9E+09,9E+09,9E+09]];
    CONST robtarget Target_90:=[[1214.248749073,634.586632651,125.675531393],[-0.000000415,0.665855066,0.746081116,-0.000000369],[-1,-1,-1,0],[2576,9E+09,9E+09,9E+09,9E+09,9E+09]];
    CONST robtarget Target_100:=[[3497.537558709,2461.137574088,1454.456324659],[0.499910434,-0.000030722,0.866077108,0.000017733],[-1,0,0,0],[3864,9E+09,9E+09,9E+09,9E+09,9E+09]];
    CONST robtarget Target_110:=[[2296.393634059,1259.823204631,1454.457605169],[0.353502598,0.612386895,0.61243072,-0.353478172],[-2,0,-1,0],[3864,9E+09,9E+09,9E+09,9E+09,9E+09]];
    CONST robtarget Target_120:=[[2206.874696407,752.235668484,670.486496878],[0.017948495,0.725103073,0.688146552,-0.018913192],[-2,0,-1,0],[3864,9E+09,9E+09,9E+09,9E+09,9E+09]];
    CONST robtarget Target_130:=[[2220.886553354,730.823804924,108.377049437],[0.008536388,0.722284375,0.691486003,-0.008917364],[-2,0,-1,0],[3864,9E+09,9E+09,9E+09,9E+09,9E+09]];
    CONST robtarget Target_140:=[[320.362651878,590.220926433,1248.380315747],[0.288561668,0.19840406,0.92517207,-0.146371558],[0,-1,0,0],[5940.941810608,9E+09,9E+09,9E+09,9E+09,9E+09]];
    CONST robtarget Target_150:=[[482.173909812,554.160304297,974.085021454],[0.197139254,0.193056634,0.951606203,-0.13531772],[0,-1,0,0],[5940.941810608,9E+09,9E+09,9E+09,9E+09,9E+09]];
    CONST robtarget Target_160:=[[618.809491746,569.611457724,770.147993108],[0.197436892,0.577373427,0.749631573,-0.256341773],[0,-1,0,0],[5940.941891889,9E+09,9E+09,9E+09,9E+09,9E+09]];
    CONST robtarget Target_170:=[[616.446518284,546.325086618,121.601414595],[0.008996777,0.049510502,0.998731596,-0.001722413],[0,0,-1,0],[5940.941810608,9E+09,9E+09,9E+09,9E+09,9E+09]];
    CONST robtarget Target_140_1:=[[-1018.09,-454.344860963,1248.38012784],[0.197436892,0.577373427,0.749631573,-0.256341773],[0,-1,-1,0],[5940.941891889,9E+09,9E+09,9E+09,9E+09,9E+09]];
    CONST robtarget Target_150_1:=[[319.209410078,535.204648154,1248.38012784],[0.197436892,0.577373427,0.749631573,-0.256341773],[0,-1,0,0],[5940.941891889,9E+09,9E+09,9E+09,9E+09,9E+09]];
    CONST robtarget Target_190:=[[673.966840107,569.60408433,1401.424579827],[0.453921347,-0.062153492,0.88883608,-0.007923214],[1,0,-1,0],[4722.757374357,9E+09,9E+09,9E+09,9E+09,9E+09]];
    CONST robtarget Target_200:=[[1073.410031722,523.80807872,67.771133201],[0.001904415,-0.052345302,0.998627132,0.000439161],[1,0,-1,0],[4722.757374357,9E+09,9E+09,9E+09,9E+09,9E+09]];
    CONST robtarget Target_210:=[[659.548293684,709.84598075,1659.5],[0.699339824,0.104517037,0.699339824,-0.104517037],[0,0,-1,0],[2382.533108305,9E+09,9E+09,9E+09,9E+09,9E+09]];
    CONST robtarget Target_220:=[[328.737767828,733.470465941,700.1000485],[0.238246517,0.168490117,0.955554758,-0.042009297],[0,0,-1,0],[2382.533108305,9E+09,9E+09,9E+09,9E+09,9E+09]];
    CONST robtarget Target_220_2:=[[328.737767828,733.470465941,181.285833737],[0.106820622,-0.001392364,0.988147783,-0.110233279],[0,-1,-1,0],[2382.533108305,9E+09,9E+09,9E+09,9E+09,9E+09]];
    CONST robtarget Target_220_2_2:=[[306.374057665,550.84910037,181.285833737],[0.106820622,-0.001392364,0.988147783,-0.110233279],[0,-1,0,0],[2382.533108305,9E+09,9E+09,9E+09,9E+09,9E+09]];
    CONST robtarget Target_90_2:=[[1214.248588097,634.586639257,-24.324468607],[-0.000000415,0.665855066,0.746081116,-0.000000369],[-1,-1,-1,0],[2576,9E+09,9E+09,9E+09,9E+09,9E+09]];
    CONST robtarget Target_90_diA:=[[1214.248566633,634.586640137,-44.324468607],[-0.000000415,0.665855066,0.746081116,-0.000000369],[-1,-1,-1,0],[2576,9E+09,9E+09,9E+09,9E+09,9E+09]];
    CONST robtarget Target_130_diA:=[[2220.488374257,721.698175201,-261.510182481],[0.008536388,0.722284375,0.691486003,-0.008917364],[-2,0,-1,0],[3864,9E+09,9E+09,9E+09,9E+09,9E+09]];
    CONST robtarget Target_200_upp:=[[1072.282744236,523.485131559,367.768841406],[0.001904415,-0.052345302,0.998627132,0.000439161],[1,0,-1,0],[4722.757374357,9E+09,9E+09,9E+09,9E+09,9E+09]];
    CONST robtarget Target_250:=[[1688.117837391,817.94570867,855.398895741],[0,0.707106781,0.707106781,0],[0,0,0,0],[0,9E+09,9E+09,9E+09,9E+09,9E+09]];
    CONST robtarget Target_230:=[[449.998,200,118.372549078],[0,0.707106781,0.707106781,0],[0,0,0,0],[6255.101552804,9E+09,9E+09,9E+09,9E+09,9E+09]];
    CONST robtarget Target_240:=[[2199.998,200,96.987347496],[0,0.707106781,0.707106781,0],[0,0,0,0],[6255.101552804,9E+09,9E+09,9E+09,9E+09,9E+09]];
    CONST robtarget Target_Wheel_R_B:=[[447.742913429,199.084023572,151.598189107],[0.000687937,-0.709243643,-0.704306869,-0.030410791],[0,0,1,0],[6547.959,9E+09,9E+09,9E+09,9E+09,9E+09]];
    CONST robtarget Target_260:=[[925.097043697,1176.228,813.889360922],[0.242436354,0.696473304,-0.664247405,0.122167661],[0,-1,0,0],[5940.942,9E+09,9E+09,9E+09,9E+09,9E+09]];
    CONST robtarget Target_270:=[[3040.792500895,1299.359973336,1454.481758418],[0.391314758,0.539089282,0.677777877,-0.311243724],[-1,0,0,0],[4322.96212259,9E+09,9E+09,9E+09,9E+09,9E+09]];
    CONST robtarget Target_Wheel_R_F:=[[2197.181,198.14,144.786550758],[0,0.707106781,0.707106781,0],[-1,1,0,0],[6237.6495745,9E+09,9E+09,9E+09,9E+09,9E+09]];
    CONST robtarget Target_Wheel_R_Pri_F:=[[1338.663941054,1043.043240219,459.467267443],[0.15653063,0.676506274,-0.691149332,0.200374712],[0,-1,0,0],[6237.6495745,9E+09,9E+09,9E+09,9E+09,9E+09]];
    CONST robtarget Target_280:=[[3091.38099561,694.76292413,831.71146423],[0.391314758,0.539089282,0.677777877,-0.311243724],[-1,0,0,0],[4322.96212259,9E+09,9E+09,9E+09,9E+09,9E+09]];
    CONST robtarget Target_290:=[[3081.730998107,658.807638145,263.483714825],[-0.000000377,0.707081698,0.707131864,-0.000000377],[-1,-1,0,0],[4322.96212259,9E+09,9E+09,9E+09,9E+09,9E+09]];
    CONST robtarget Target_Tool_Axel_last:=[[3081.730784907,658.80763813,63.483714825],[-0.000000377,0.707081698,0.707131864,-0.000000377],[-1,-1,0,0],[4322.96212259,9E+09,9E+09,9E+09,9E+09,9E+09]];
    CONST robtarget Target_Tool_Axel_R_last:=[[3081.730786484,658.80763813,64.963510663],[-0.000000377,0.707081698,0.707131864,-0.000000377],[-1,-1,0,0],[4322.96212259,9E+09,9E+09,9E+09,9E+09,9E+09]];
    CONST robtarget Target_300:=[[3782.656138088,1331.060088619,1403.237411059],[0.195338848,0.633678409,0.729016058,-0.16979398],[-1,0,-1,0],[5175,9E+09,9E+09,9E+09,9E+09,9E+09]];
    CONST robtarget Target_310:=[[3871.292586337,700.699290974,849.981871233],[0.039499264,0.655133169,0.753698538,-0.034334425],[-1,-1,0,0],[5175,9E+09,9E+09,9E+09,9E+09,9E+09]];
    CONST robtarget Target_320:=[[3666.244896019,658.849107068,169.096091733],[0.039499264,0.655133169,0.753698538,-0.034334425],[-1,0,-1,0],[5175,9E+09,9E+09,9E+09,9E+09,9E+09]];
    CONST robtarget Target_Tool_ArmP_R_last:=[[3666.244682819,658.849107053,-30.903908267],[0.039499264,0.655133169,0.753698538,-0.034334425],[-1,0,-1,0],[5175,9E+09,9E+09,9E+09,9E+09,9E+09]];
    CONST robtarget Target_330:=[[-21.35697429,664.114103086,1268.967612304],[0.120017866,0.172353755,0.97746716,-0.021162394],[0,0,-1,0],[2486.201455697,9E+09,9E+09,9E+09,9E+09,9E+09]];
    CONST robtarget Target_340:=[[109.386903746,693.94582789,1039.665090814],[-0.000000001,0.173648102,0.984807766,0.000000007],[0,0,-1,0],[2486.201455697,9E+09,9E+09,9E+09,9E+09,9E+09]];
    CONST robtarget Target_350:=[[109.048,571.763342709,772.223228929],[-0.000000001,0.173648102,0.984807766,0.000000007],[0,0,-1,0],[2486.201455697,9E+09,9E+09,9E+09,9E+09,9E+09]];
    CONST robtarget Target_AxP_tR_R_Last:=[[109.048,571.763342709,572.223228929],[-0.000000001,0.173648102,0.984807766,0.000000007],[0,0,-1,0],[2486.201,9E+09,9E+09,9E+09,9E+09,9E+09]];
    CONST robtarget Target_360:=[[147.015240636,559.016761098,1131.994072821],[0.106034295,0.347956188,0.93065113,-0.039644601],[0,-1,-1,0],[575.958714265,9E+09,9E+09,9E+09,9E+09,9E+09]];
    CONST robtarget Target_370:=[[134.666658073,569.751220324,814.763311248],[0.057182476,-0.349554164,-0.93492511,-0.021379653],[0,0,-1,0],[575.958714265,9E+09,9E+09,9E+09,9E+09,9E+09]];
    CONST robtarget Target_380:=[[71.457,593.548550758,349.980925618],[0.007473756,0.347245371,0.936642376,0.045451685],[0,0,-1,0],[575.958714265,9E+09,9E+09,9E+09,9E+09,9E+09]];
    CONST robtarget Target_ArmP_tR_R_Last:=[[71.457,593.548550758,149.980925618],[0.007473756,0.347245371,0.936642376,0.045451685],[0,0,-1,0],[575.958714265,9E+09,9E+09,9E+09,9E+09,9E+09]];
    CONST robtarget Target_390:=[[925.097043697,1176.228,813.889360922],[0.242436354,0.696473304,-0.664247405,0.122167661],[0,-1,0,0],[5940.942,9E+09,9E+09,9E+09,9E+09,9E+09]];
    CONST robtarget Target_AxlP_tT_Right_Pre:=[[1338.869,371.254701034,1810.868145602],[0.047032358,0.705540897,-0.705540897,0.047032358],[0,0,-1,0],[5034.183673469,9E+09,9E+09,9E+09,9E+09,9E+09]];
    CONST robtarget Target_AxlP_tT_Right_Pre_F:=[[2216.362,213.985,1122.693550758],[0,0.707106781,0.707106781,0],[-1,-1,2,0],[5530,9E+09,9E+09,9E+09,9E+09,9E+09]];
    CONST robtarget Target_AxlP_tT_Right_F:=[[2216.362,213.985,222.693550758],[0,0.707106781,0.707106781,0],[-1,-1,2,0],[5949.489795918,9E+09,9E+09,9E+09,9E+09,9E+09]];
    CONST robtarget Target_AxlP_tT_Right_Pre_B:=[[450.122,193.774,1116.772550758],[0,0.707106781,0.707106781,0],[0,0,1,0],[5530,9E+09,9E+09,9E+09,9E+09,9E+09]];
    CONST robtarget Target_AxlP_tT_Right_B:=[[450.122,193.774,216.772550758],[0,0.707106781,0.707106781,0],[0,0,1,0],[6350.321542907,9E+09,9E+09,9E+09,9E+09,9E+09]];
    CONST robtarget Target_Link_tT_Right_Pre:=[[1354.222,827.860897308,1547.552022339],[0.055478959,0.704927007,-0.704927007,0.055478959],[0,-3,2,0],[5034.183673469,9E+09,9E+09,9E+09,9E+09,9E+09]];
    CONST robtarget Target_Link_tT_Right_Pre_:=[[1680.933,243.392,479.815550758],[0,0.707106781,0.707106781,0],[-1,-1,2,0],[5994.114762066,9E+09,9E+09,9E+09,9E+09,9E+09]];
    CONST robtarget Target_Link_tT_Right:=[[1680.933,243.392,279.815550758],[0,0.707106781,0.707106781,0],[-1,-1,2,0],[5994.114762066,9E+09,9E+09,9E+09,9E+09,9E+09]];
    CONST robtarget Target_Link_tT_Right_Pre_Last:=[[1680.933,243.392,479.815550758],[0,0,1,0],[-1,-3,3,0],[5994.114762066,9E+09,9E+09,9E+09,9E+09,9E+09]];
    CONST robtarget Target_Link_tT_Right_last:=[[1680.933,243.392,279.815550758],[0,-0.069756474,0.99756405,0],[-1,-3,3,0],[5994.114762066,9E+09,9E+09,9E+09,9E+09,9E+09]];
    CONST robtarget Target_ArmP_tT_Right_Pre:=[[1338.868999791,767.291108113,1563.727110087],[0.061628481,0.704416021,-0.704416021,0.061628481],[0,0,-1,0],[5034.183673469,9E+09,9E+09,9E+09,9E+09,9E+09]];
    CONST robtarget Target_ArmP_tT_Right_Pre_Last_B:=[[793.248,246.837,633.596207225],[0,0.707106781,0.707106781,0],[0,0,1,0],[6186.102175139,9E+09,9E+09,9E+09,9E+09,9E+09]];
    CONST robtarget Target_ArmP_tT_Right_Last_B:=[[793.248,246.837,333.596207225],[0,0.707106781,0.707106781,0],[0,0,1,0],[6186.102175139,9E+09,9E+09,9E+09,9E+09,9E+09]];
    CONST robtarget Target_ArmP_tT_Right_Pre_Last_F:=[[2552.837,242.052,627.194550758],[0,0.707106781,0.707106781,0],[-1,-1,2,0],[6360.634088471,9E+09,9E+09,9E+09,9E+09,9E+09]];
    CONST robtarget Target_ArmP_tT_Right_Last_F:=[[2552.837,242.052,327.194550758],[0,0.707106781,0.707106781,0],[-1,-1,2,0],[6360.634088471,9E+09,9E+09,9E+09,9E+09,9E+09]];
    CONST robtarget Target_Wheel_R_Pre_Last_F:=[[2197.181,198.14,344.786550758],[0,0.707106781,0.707106781,0],[-1,1,0,0],[6237.6495745,9E+09,9E+09,9E+09,9E+09,9E+09]];
    CONST robtarget Target_Wheel_R_Pre_F:=[[1338.663941054,1043.043240219,459.467267443],[0.15653063,0.676506274,-0.691149332,0.200374712],[0,-1,0,0],[6237.6495745,9E+09,9E+09,9E+09,9E+09,9E+09]];
    CONST robtarget Target_Wheel_R_Last_F:=[[2197.181,198.14,144.786550758],[0,0.707106781,0.707106781,0],[-1,1,0,0],[6237.6495745,9E+09,9E+09,9E+09,9E+09,9E+09]];
    CONST robtarget Target_Wheel_R_Last_B:=[[447.742913429,199.084023572,151.598189107],[0.000687937,-0.709243643,-0.704306869,-0.030410791],[0,-2,-1,0],[6547.959,9E+09,9E+09,9E+09,9E+09,9E+09]];
    CONST robtarget Target_Wheel_R_Pre_Last_B:=[[447.742913429,199.084023572,351.598189107],[0.000687937,-0.709243643,-0.704306869,-0.030410791],[0,-2,-1,0],[6547.959,9E+09,9E+09,9E+09,9E+09,9E+09]];
!***********************************************************
    !
    ! Module:  Module1
    !
    ! Description:
    !   <Insert description here>
    !
    ! Author: haba0028
    !
    ! Version: 1.0
    !
    !***********************************************************


    !***********************************************************
    !
    ! Procedure main
    !
    !   This is the entry point of your program
    !
    !***********************************************************
    PROC main()
        !Add your code here
        SetDO diAttachTool,0;
        SetDO doAtWhRi,0;
        SetDO doAttachTo_S,0;
        SetDO Att_link,0;

!        Path_Attach_Tool_Stack_Right;
!        Path_diAttach_Tool_Stack_Right;
!        Path_Attach_Stack;

!        Path_Attach_Tool_Link_Right;
!        Path_Attach_Link;
!        Path_diAttach_Tool_Link_Right;


!        Path_Attach_Tool_Wheel_Right;
!        Path_Attach_wheel;
!        Path_Att_Wh_Train_Right_2;
!        Path_Attach_wheel;
!        Path_Att_Wh_Train_Right_1;
!        Path_diAttach_Tool_Wheel_Right;




!! That Works:

        Path_Attach_Tool_Wheel_Right;
        Path_At_Wh_tR_Right;
        Path_Att_Wh_tT_Right_F;
        Path_At_Wh_tR_Right;
        Path_Att_Wh_tT_Right_B;
        Path_diAttach_Tool_Wheel_Right;

        Path_Attach_Tool_AxelP_tR_Right;
        Path_Att_AxlP_tR_Right;
        Path_At_AxlP_tT_R_F;
        Path_Att_AxlP_tR_Right;
        Path_At_AxlP_tT_R_B;
        Path_diAttac_Tool_AxelP_tR_Right;


        Path_Attach_Tool_Link_Right;
        Path_Attach_Link_tR_Right;
        Path_At_Link_tT_R;
        Path_diAttach_Tool_Link_Right;

        Path_Attach_Tool_ArmP_tR_Right;
        Path_Att_ArmP_tR_Right;
        Path_At_ArmP_tT_R_F;
        Path_Att_ArmP_tR_Right;
        Path_At_ArmP_tT_R_B;
        Path_diAttach_Tool_ArmP_tR_Right;

    ENDPROC




    !! Attach/diAttach Tools To Robot
    PROC Path_Attach_Tool_Wheel_Right()
        WaitTime 0.4;
        MoveJ Target_110,v500,fine,tool0\WObj:=stand_tool_Right;
        MoveL Target_120,v500,fine,tool0\WObj:=stand_tool_Right;
        MoveL Target_130,v500,fine,tool0\WObj:=stand_tool_Right;
        WaitTime 0.3;
        SetDO doAttachTo_S,1;
        WaitTime 0.3;
        MoveL Target_120,v500,fine,Tool_Wheel\WObj:=stand_tool_Right;
        MoveL Target_110,v500,fine,Tool_Wheel\WObj:=stand_tool_Right;
    ENDPROC
    PROC Path_diAttach_Tool_Wheel_Right()
        WaitTime 0.4;
        MoveJ Target_110,v500,fine,Tool_Wheel\WObj:=stand_tool_Right;
        MoveL Target_120,v500,fine,Tool_Wheel\WObj:=stand_tool_Right;
        MoveL Target_130,v500,fine,tool0\WObj:=stand_tool_Right;
        WaitTime 0.3;
        SetDO doAttachTo_S,0;
        WaitTime 0.3;
        MoveL Target_120,v500,fine,tool0\WObj:=stand_tool_Right;
        MoveL Target_110,v500,fine,tool0\WObj:=stand_tool_Right;
    ENDPROC

    PROC Path_Attach_Tool_Link_Right()
        MoveJ Target_70,v500,fine,tool0\WObj:=stand_tool_Right;
        MoveL Target_80,v500,fine,tool0\WObj:=stand_tool_Right;
        MoveL Target_90,v500,fine,tool0\WObj:=stand_tool_Right;
        WaitTime 0.3;
!        SetDO diAttachTool,1;
        SetDO doAttachTo_S,1;
        WaitTime 0.3;
        MoveL Target_80,v500,fine,Tool_Link\WObj:=stand_tool_Right;
        MoveL Target_70,v500,fine,Tool_Link\WObj:=stand_tool_Right;
    ENDPROC
    PROC Path_diAttach_Tool_Link_Right()
        MoveJ Target_70,v500,fine,Tool_Link\WObj:=stand_tool_Right;
        MoveL Target_80,v500,fine,Tool_Link\WObj:=stand_tool_Right;
        MoveL Target_90,v500,fine,tool0\WObj:=stand_tool_Right;
        WaitTime 0.3;
!        SetDO diAttachTool,0;
        SetDO doAttachTo_S,0;
        WaitTime 0.3;
        MoveL Target_80,v500,fine,tool0\WObj:=stand_tool_Right;
        MoveL Target_70,v500,fine,tool0\WObj:=stand_tool_Right;
    ENDPROC

    PROC Path_Attach_Tool_Stack_Right()
        MoveJ Target_30,v500,fine,tool0\WObj:=stand_tool_Right;
        MoveL Target_20,v500,fine,tool0\WObj:=stand_tool_Right;
        MoveL Target_10,v500,fine,tool0\WObj:=stand_tool_Right;
        WaitTime 0.3;
!        SetDO diAttachTool,1;
        SetDO doAttachTo_S,1;
        WaitTime 0.3;
        MoveL Target_20,v500,fine,tool0\WObj:=stand_tool_Right;
        MoveL Target_30,v500,fine,tool0\WObj:=stand_tool_Right;
    ENDPROC
    PROC Path_diAttach_Tool_Stack_Right()
        MoveJ Target_30,v500,fine,tool0\WObj:=stand_tool_Right;
        MoveL Target_20,v500,fine,tool0\WObj:=stand_tool_Right;
        MoveL Target_10,v500,fine,tool0\WObj:=stand_tool_Right;
        WaitTime 0.3;
!        SetDO diAttachTool,0;
        SetDO doAttachTo_S,0;
        WaitTime 0.3;
        MoveL Target_20,v500,fine,Tool_Stack\WObj:=stand_tool_Right;
        MoveL Target_30,v500,fine,Tool_Stack\WObj:=stand_tool_Right;
    ENDPROC

    PROC Path_Attach_Tool_AxelP_tR_Right()
        MoveJ Target_270,v500,fine,tool0\WObj:=stand_tool_Right;
        MoveL Target_280,v500,fine,tool0\WObj:=stand_tool_Right;
        MoveL Target_290,v500,fine,tool0\WObj:=stand_tool_Right;
        MoveL Target_Tool_Axel_R_last,v500,fine,tool0\WObj:=stand_tool_Right;
        WaitTime 0.3;
!        SetDO diAttachTool,1;
        SetDO doAttachTo_S,1;
        WaitTime 1;
        MoveL Target_290,v500,fine,Tool_Axelpin\WObj:=stand_tool_Right;
        MoveL Target_280,v500,fine,Tool_Axelpin\WObj:=stand_tool_Right;
        MoveL Target_270,v500,fine,Tool_Axelpin\WObj:=stand_tool_Right;
    ENDPROC

    PROC Path_diAttac_Tool_AxelP_tR_Right()
        WaitTime 0.4;
        MoveJ Target_270,v500,fine,tool0\WObj:=stand_tool_Right;
        MoveL Target_280,v500,fine,tool0\WObj:=stand_tool_Right;
        MoveL Target_290,v500,fine,tool0\WObj:=stand_tool_Right;
        MoveL Target_Tool_Axel_R_last,v500,fine,tool0\WObj:=stand_tool_Right;
        WaitTime 0.3;
!        SetDO diAttachTool,1;
        SetDO doAttachTo_S,0;
        WaitTime 1;
        MoveL Target_290,v500,fine,Tool_Axelpin\WObj:=stand_tool_Right;
        MoveL Target_280,v500,fine,Tool_Axelpin\WObj:=stand_tool_Right;
        MoveL Target_270,v500,fine,Tool_Axelpin\WObj:=stand_tool_Right;
    ENDPROC

    PROC Path_Attach_Tool_ArmP_tR_Right()
        WaitTime 0.4;
        MoveJ Target_300,v500,fine,tool0\WObj:=stand_tool_Right;
        MoveL Target_310,v500,fine,tool0\WObj:=stand_tool_Right;
        MoveL Target_320,v500,fine,tool0\WObj:=stand_tool_Right;
        MoveL Target_Tool_ArmP_R_last,v500,fine,tool0\WObj:=stand_tool_Right;
        WaitTime 0.3;
!        SetDO diAttachTool,1;
        SetDO doAttachTo_S,1;
        WaitTime 1;
        MoveL Target_320,v500,fine,Tool_ArmPin\WObj:=stand_tool_Right;
        MoveL Target_310,v500,fine,Tool_ArmPin\WObj:=stand_tool_Right;
        MoveL Target_300,v500,fine,Tool_ArmPin\WObj:=stand_tool_Right;
    ENDPROC

    PROC Path_diAttach_Tool_ArmP_tR_Right()
        WaitTime 0.4;
        MoveJ Target_300,v500,fine,tool0\WObj:=stand_tool_Right;
        MoveL Target_310,v500,fine,tool0\WObj:=stand_tool_Right;
        MoveL Target_320,v500,fine,tool0\WObj:=stand_tool_Right;
        MoveL Target_Tool_ArmP_R_last,v500,fine,tool0\WObj:=stand_tool_Right;
        WaitTime 0.3;
!        SetDO diAttachTool,1;
        SetDO doAttachTo_S,0;
        WaitTime 1;
        MoveL Target_320,v500,fine,Tool_ArmPin\WObj:=stand_tool_Right;
        MoveL Target_310,v500,fine,Tool_ArmPin\WObj:=stand_tool_Right;
        MoveL Target_300,v500,fine,Tool_ArmPin\WObj:=stand_tool_Right;
    ENDPROC













    !! Attach Parts to the Tolls in Robots
    PROC Path_At_Wh_tR_Right()
        WaitTime 0.4;
        MoveJ Target_140,v500,fine,Tool_Wheel\WObj:=InFeWOb_Right_1;
        MoveL Target_150,v500,fine,Tool_Wheel\WObj:=InFeWOb_Right_1;
        MoveL Target_170,v500,fine,Tool_Wheel\WObj:=InFeWOb_Right_1;
        WaitTime 0.4;
        SetDO doAtWhRi,1;
        WaitTime 1;
        MoveL Target_150,v500,fine,Tool_Wheel\WObj:=InFeWOb_Right_1;
        MoveL Target_140,v500,fine,Tool_Wheel\WObj:=InFeWOb_Right_1;
    ENDPROC

    PROC Path_Attach_Link_tR_Right()
        WaitTime 0.4;
        MoveJ Target_190,v500,fine,Tool_Link\WObj:=InFeWOb_Right_2;
        MoveL Target_200_upp,v500,fine,Tool_Wheel\WObj:=InFeWOb_Right_2;
        MoveJ Target_200,v500,fine,Tool_Link\WObj:=InFeWOb_Right_2;
        WaitTime 0.4;
        SetDO Att_link,1;
        WaitTime 1;
        MoveL Target_200_upp,v500,fine,Tool_Wheel\WObj:=InFeWOb_Right_2;
        MoveJ Target_190,v500,fine,Tool_Link\WObj:=InFeWOb_Right_2;
    ENDPROC

    PROC Path_Att_AxlP_tR_Right()
        WaitTime 0.4;
        MoveJ Target_330,v500,fine,Tool_Axelpin\WObj:=InFeWOb_Right_3;
        MoveL Target_340,v500,fine,Tool_Axelpin\WObj:=InFeWOb_Right_3;
        MoveL Target_350,v500,fine,Tool_Axelpin\WObj:=InFeWOb_Right_3;
        MoveL Target_AxP_tR_R_Last,v500,fine,Tool_Axelpin\WObj:=InFeWOb_Right_3;
        WaitTime 0.4;
        SetDO doAt_AxelP_Right,1;
        WaitTime 1;
        MoveL Target_350,v500,fine,Tool_Axelpin\WObj:=InFeWOb_Right_3;
        MoveL Target_340,v500,fine,Tool_Axelpin\WObj:=InFeWOb_Right_3;
        MoveL Target_330,v500,fine,Tool_Axelpin\WObj:=InFeWOb_Right_3;
    ENDPROC

    PROC Path_Att_ArmP_tR_Right()
        WaitTime 0.4;
        MoveJ Target_360,v500,fine,Tool_ArmPin\WObj:=InFeWOb_Right_4;
        MoveL Target_370,v500,fine,Tool_ArmPin\WObj:=InFeWOb_Right_4;
        MoveL Target_380,v500,fine,Tool_ArmPin\WObj:=InFeWOb_Right_4;
        MoveL Target_ArmP_tR_R_Last,v500,fine,Tool_ArmPin\WObj:=InFeWOb_Right_4;
        WaitTime 0.4;
        SetDO doAt_ArmP_Right,1;
        WaitTime 1;
        MoveL Target_380,v500,fine,Tool_ArmPin\WObj:=InFeWOb_Right_4;
        MoveL Target_370,v500,fine,Tool_ArmPin\WObj:=InFeWOb_Right_4;
        MoveL Target_360,v500,fine,Tool_ArmPin\WObj:=InFeWOb_Right_4;
    ENDPROC





    !! Attach Parts to the Train
    PROC Path_Att_Wh_tT_Right_F()
        WaitTime 0.4;
        MoveJ Target_390,v500,fine,Tool_Wheel\WObj:=TrRiFcWOb;
        MoveL Target_Wheel_R_Pre_F,v500,fine,Tool_Wheel\WObj:=TrRiFcWOb;
        MoveL Target_Wheel_R_Pre_Last_F,v500,fine,Tool_Wheel\WObj:=TrRiFcWOb;
        MoveL Target_Wheel_R_Last_F,v500,fine,Tool_Wheel\WObj:=TrRiFcWOb;
        WaitTime 0.4;
        SetDO doAtWhRi,0;
        WaitTime 1;
        MoveL Target_Wheel_R_Pre_Last_F,v500,fine,Tool_Wheel\WObj:=TrRiFcWOb;
        MoveL Target_Wheel_R_Pre_F,v500,fine,Tool_Wheel\WObj:=TrRiFcWOb;
    ENDPROC

    PROC Path_Att_Wh_tT_Right_B()
        WaitTime 0.4;
        MoveJ Target_390,v500,fine,Tool_Wheel\WObj:=TrRiFcWOb;
        MoveL Target_Wheel_R_Pre_Last_B,v500,fine,Tool_Wheel\WObj:=TrRiFcWOb;
        MoveL Target_Wheel_R_Last_B,v500,fine,Tool_Wheel\WObj:=TrRiFcWOb;
        WaitTime 0.4;
        SetDO doAtWhRi,0;
        WaitTime 1;
        MoveL Target_Wheel_R_Pre_Last_B,v500,fine,Tool_Wheel\WObj:=TrRiFcWOb;
        MoveL Target_390,v500,fine,Tool_Wheel\WObj:=TrRiFcWOb;
    ENDPROC


    PROC Path_At_AxlP_tT_R_F()
        WaitTime 0.4;
        MoveJ Target_AxlP_tT_Right_Pre,v500,fine,Tool_Axelpin\WObj:=TrRiFcWOb;
        MoveL Target_AxlP_tT_Right_Pre_F,v500,fine,Tool_Axelpin\WObj:=TrRiFcWOb;
        MoveL Target_AxlP_tT_Right_F,v500,fine,Tool_Axelpin\WObj:=TrRiFcWOb;
        WaitTime 0.4;
        SetDO doAt_AxelP_Right,0;
        WaitTime 1;
        MoveL Target_AxlP_tT_Right_Pre_F,v500,fine,Tool_Axelpin\WObj:=TrRiFcWOb;
        MoveL Target_AxlP_tT_Right_Pre,v500,fine,Tool_Axelpin\WObj:=TrRiFcWOb;
    ENDPROC
    PROC Path_At_AxlP_tT_R_B()
        WaitTime 0.4;
        MoveJ Target_AxlP_tT_Right_Pre,v500,fine,Tool_Axelpin\WObj:=TrRiFcWOb;
        MoveL Target_AxlP_tT_Right_Pre_B,v500,fine,Tool_Axelpin\WObj:=TrRiFcWOb;
        MoveL Target_AxlP_tT_Right_B,v500,fine,Tool_Axelpin\WObj:=TrRiFcWOb;
        WaitTime 0.4;
        SetDO doAt_AxelP_Right,0;
        MoveL Target_AxlP_tT_Right_Pre_B,v500,fine,Tool_Axelpin\WObj:=TrRiFcWOb;
        MoveL Target_AxlP_tT_Right_Pre,v500,fine,Tool_Axelpin\WObj:=TrRiFcWOb;
    ENDPROC


    PROC Path_At_Link_tT_R()
        WaitTime 0.4;
        MoveJ Target_Link_tT_Right_Pre,v500,fine,Tool_Link\WObj:=TrRiFcWOb;
        MoveL Target_Link_tT_Right_Pre_Last,v500,fine,Tool_Link\WObj:=TrRiFcWOb;
        MoveL Target_Link_tT_Right_last,v500,fine,Tool_Link\WObj:=TrRiFcWOb;
        WaitTime 0.4;
        SetDO Att_link,0;
        WaitTime 1;
        MoveL Target_Link_tT_Right_Pre_Last,v500,fine,Tool_Link\WObj:=TrRiFcWOb;
        MoveL Target_Link_tT_Right_Pre,v500,fine,Tool_Link\WObj:=TrRiFcWOb;
    ENDPROC

    PROC Path_At_ArmP_tT_R_B()
        WaitTime 0.4;
        MoveJ Target_ArmP_tT_Right_Pre,v500,fine,Tool_ArmPin\WObj:=TrRiFcWOb;
        MoveL Target_ArmP_tT_Right_Pre_Last_B,v500,fine,Tool_ArmPin\WObj:=TrRiFcWOb;
        MoveL Target_ArmP_tT_Right_Last_B,v500,fine,Tool_ArmPin\WObj:=TrRiFcWOb;
        WaitTime 1;
        WaitTime 0.4;
        SetDO doAt_ArmP_Right,0;
        WaitTime 1;
        MoveL Target_ArmP_tT_Right_Pre_Last_B,v500,fine,Tool_ArmPin\WObj:=TrRiFcWOb;
        MoveL Target_ArmP_tT_Right_Pre,v500,fine,Tool_ArmPin\WObj:=TrRiFcWOb;
    ENDPROC
    PROC Path_At_ArmP_tT_R_F()
        WaitTime 0.4;
        MoveJ Target_ArmP_tT_Right_Pre,v500,fine,Tool_ArmPin\WObj:=TrRiFcWOb;
        MoveL Target_ArmP_tT_Right_Pre_Last_F,v500,fine,Tool_ArmPin\WObj:=TrRiFcWOb;
        MoveL Target_ArmP_tT_Right_Last_F,v500,fine,Tool_ArmPin\WObj:=TrRiFcWOb;
        WaitTime 1;
        WaitTime 0.4;
        SetDO doAt_ArmP_Right,0;
        WaitTime 1;
        MoveL Target_ArmP_tT_Right_Pre_Last_F,v500,fine,Tool_ArmPin\WObj:=TrRiFcWOb;
        MoveL Target_ArmP_tT_Right_Pre,v500,fine,Tool_ArmPin\WObj:=TrRiFcWOb;
    ENDPROC


ENDMODULE

